(* IEC 61131-3 sources: Elmo_Master/test/Reports_Lasal/C78_20260807_publish_split_rebaseline (part 5) *)

	homePreemptionResult := CopyAxisOwnershipPreemption(
			PreemptedAdmissionToken:=homeAdmissionToken,
			PreemptedOwnerGeneration:=homeOwnerGeneration,
			pDest:=#homePreemptionSnapshot[0],
			DestSize:=sizeof(homePreemptionSnapshot));
	if (homePreemptionResult >= LMC_OWNER_PREEMPT_STATUS_PENDING_FREEZE) &
		   (homePreemptionResult <=
		    LMC_OWNER_PREEMPT_STATUS_CLEANUP_QUARANTINED) then
		homePreemptionSnapshotValid :=
				(homePreemptionSnapshot[0]$UDINT =
				 LMC_OWNER_PREEMPT_COPY_MAGIC) &
				(homePreemptionSnapshot[4]$UDINT =
				 LMC_OWNER_IDENTITY_VERSION) &
				(homePreemptionSnapshot[8]$UDINT =
				 LMC_OWNER_PREEMPT_COPY_HEADER_BYTES) &
				(homePreemptionSnapshot[12]$UDINT =
				 sizeof(homePreemptionSnapshot)) &
				(homePreemptionSnapshot[16]$DINT = homePreemptionResult) &
				(homePreemptionSnapshot[32]$UDINT =
				 homeAxisMask) &
				(homePreemptionSnapshot[36]$UDINT =
				 homeAdmissionToken) &
				(homePreemptionSnapshot[40]$UDINT =
				 homeOwnerGeneration) &
				(homePreemptionSnapshot[44]$UDINT =
				 homeSessionEpoch) &
				(homePreemptionSnapshot[48]$UDINT =
				 homeRequestSequence) &
				(homePreemptionSnapshot[52]$UDINT = 0x7D13) &
				(homePreemptionSnapshot[56]$DINT = ZeroHomeState[9]) &
				(homePreemptionSnapshot[60]$DINT =
				 LMC_OWNER_KIND_LMC_HOME) &
				(homePreemptionSnapshot[64]$DINT =
				 LMC_OWNER_RESOURCE_LMC_HOME_ENGINE) &
				(homePreemptionSnapshot[68]$DINT =
				 LMC_OWNER_ADMISSION_LIFECYCLE) &
				(homePreemptionSnapshot[72]$DINT =
				 LMC_OWNER_STATE_LMC_HOME_ACTIVE) &
				(homePreemptionSnapshot[76]$UDINT = 56) &
				((homePreemptionSnapshot[104]$UDINT and
				  homeAxisMask) = homeAxisMask) &
				(homePreemptionSnapshot[108]$UDINT <> 0) &
				(homePreemptionSnapshot[112]$UDINT <> 0) &
				((homePreemptionSnapshot[124]$DINT =
				  LMC_OWNER_STATE_RESERVED) |
				 (homePreemptionSnapshot[124]$DINT =
				  LMC_OWNER_STATE_SAFETY_PREEMPTING) |
				 (homePreemptionSnapshot[124]$DINT =
				  LMC_OWNER_STATE_QUARANTINED)) &
				(homePreemptionSnapshot[128]$UDINT <> 0) &
				(homePreemptionSnapshot[132]$UDINT <> 0) &
				(homePreemptionSnapshot[136]$DINT =
				 LMC_OWNER_ADMISSION_SAFETY) &
				(homePreemptionSnapshot[140]$UDINT = 0) &
				(homePreemptionSnapshot[144]$UINT = 1) &
				(homePreemptionSnapshot[146]$UINT = 0) &
				(homePreemptionSnapshot[148]$UDINT =
				 ZeroHomeState[4]$UDINT) &
				(homePreemptionSnapshot[152]$UDINT =
				 ZeroHomeState[1]$UDINT) &
				(homePreemptionSnapshot[156]$UDINT =
				 ZeroHomeState[2]$UDINT) &
				(homePreemptionSnapshot[160]$UDINT =
				 ZeroHomeState[3]$UDINT) &
				(homePreemptionSnapshot[164]$UDINT =
				 ZeroHomeState[5]$UDINT) &
				(homePreemptionSnapshot[168]$UDINT =
				 ZeroHomeState[6]$UDINT) &
				(homePreemptionSnapshot[172]$UDINT =
				 ZeroHomeState[7]$UDINT) &
				(homePreemptionSnapshot[176]$UDINT =
				 ZeroHomeState[8]$UDINT) &
				(homePreemptionSnapshot[180]$UINT =
				 TO_UINT(ZeroHomeState[10])) &
				(homePreemptionSnapshot[182]$UINT = 0) &
				(homePreemptionSnapshot[184]$DINT = ZeroHomeState[11]) &
				(homePreemptionSnapshot[188]$DINT = ZeroHomeState[12]) &
				(homePreemptionSnapshot[192]$UDINT =
				 ZeroHomeState[13]$UDINT) &
				(homePreemptionSnapshot[196]$UDINT = 0x454D4F48);
		if homePreemptionResult =
			   LMC_OWNER_PREEMPT_STATUS_PENDING_FREEZE then
			homePreemptionSnapshotValid :=
					homePreemptionSnapshotValid &
					((homePreemptionSnapshot[24]$UDINT and
					  homeAxisMask) = homeAxisMask) &
					((homePreemptionSnapshot[28]$UDINT and
					  homeAxisMask) = 0) &
					(homePreemptionSnapshot[124]$DINT =
					 LMC_OWNER_STATE_RESERVED);
		elsif homePreemptionResult =
			      LMC_OWNER_PREEMPT_STATUS_CLEANUP_REQUIRED then
			homePreemptionSnapshotValid :=
					homePreemptionSnapshotValid &
					((homePreemptionSnapshot[24]$UDINT and
					  homeAxisMask) = homeAxisMask) &
					((homePreemptionSnapshot[28]$UDINT and
					  homeAxisMask) = 0) &
					(homePreemptionSnapshot[124]$DINT <>
					 LMC_OWNER_STATE_RESERVED);
		elsif homePreemptionResult =
			      LMC_OWNER_PREEMPT_STATUS_CLEANUP_COMPLETE then
			homePreemptionSnapshotValid :=
					homePreemptionSnapshotValid &
					((homePreemptionSnapshot[28]$UDINT and
					  homeAxisMask) = homeAxisMask);
		end_if;
	end_if;

	if homePreemptionResult =
		   LMC_OWNER_PREEMPT_STATUS_PENDING_FREEZE then
		// The safety handler may run only after exact snapshot and cancel proof.
		homeFlags := homeFlags or LMC_HOME_FLAG_CANCEL_REQUIRED;
		ZeroHomeState[39] := LMC_HOME_ENGINE_CANCEL_DRAIN;
		if homePreemptionSnapshotValid &
		   (IsClientConnected(#InputLatch) <> 0) then
			homeCancelResult := InputLatch.CancelAxisZeroHome(
				OperationToken:=homeAdmissionToken);
		end_if;
		if homePreemptionSnapshotValid & (homeCancelResult >= 0) then
			if (homeFlags and LMC_HOME_FLAG_CANCEL_PUBLISHED) = 0 then
				ZeroHomeState[54]$UDINT := homeServiceNow;
			end_if;
			homeFlags := homeFlags or LMC_HOME_FLAG_CANCEL_PUBLISHED or
				LMC_HOME_FLAG_PREEMPTION_CLEANUP or
				LMC_HOME_FLAG_SAFETY_DISPATCH_READY;
		else
			ZeroHomeState[31] := homeCancelResult;
			OwnershipState[24] := 1;
		end_if;
		ZeroHomeState[56]$UDINT := homeFlags;
		RETURN;
	elsif (homePreemptionResult =
		       LMC_OWNER_PREEMPT_STATUS_CLEANUP_COMPLETE) &
		      homePreemptionSnapshotValid then
		// Exact owner cleanup replay is sufficient to finish the retained record.
		ZeroHomeState[14] := 1;
		ZeroHomeState[15] := -31000;
		ZeroHomeState[16] := 39;
		ZeroHomeState[30]$UDINT := homeServiceNow;
		ZeroHomeState[31] := -10;
		ZeroHomeState[47] := 1;
		ZeroHomeState[57] := LMC_HOME_RECORD_ABORTED;
		ZeroHomeState[58] := LMC_OWNER_REPORT_TERMINAL_SAFE_FAILURE;
		ZeroHomeState[59] := LMC_OWNER_CLEANUP_COMPLETE_SAFE;
		homeFlags := homeFlags or LMC_HOME_FLAG_CANCEL_REQUIRED or
			LMC_HOME_FLAG_CANCEL_PUBLISHED or
			LMC_HOME_FLAG_EXACT_RT_TERMINAL or
			LMC_HOME_FLAG_OWNER_FINALIZE_INTENT or
			LMC_HOME_FLAG_OWNER_FINALIZE_ACCEPTED or
			LMC_HOME_FLAG_TERMINAL_PUBLISHED or
			LMC_HOME_FLAG_PREEMPTION_CLEANUP;
		ZeroHomeState[56]$UDINT := homeFlags;
		ZeroHomeState[39] := LMC_HOME_ENGINE_TERMINAL;
		ZeroHomeState[0] := LMC_HOME_RECORD_ABORTED;
		RETURN;
	elsif (homePreemptionResult =
		       LMC_OWNER_PREEMPT_STATUS_CLEANUP_QUARANTINED) &
		      homePreemptionSnapshotValid then
		ZeroHomeState[14] := 1;
		ZeroHomeState[15] := -31000;
		ZeroHomeState[16] := 42;
		ZeroHomeState[30]$UDINT := homeServiceNow;
		ZeroHomeState[31] := -8;
		ZeroHomeState[47] := 1;
		ZeroHomeState[57] := LMC_HOME_RECORD_QUARANTINED;
		ZeroHomeState[58] := LMC_OWNER_REPORT_QUARANTINE;
		ZeroHomeState[59] := LMC_OWNER_CLEANUP_INCOMPLETE_QUARANTINE;
		homeFlags := homeFlags or LMC_HOME_FLAG_CANCEL_REQUIRED or
			LMC_HOME_FLAG_OWNER_FINALIZE_INTENT or
			LMC_HOME_FLAG_OWNER_FINALIZE_ACCEPTED or
			LMC_HOME_FLAG_TERMINAL_PUBLISHED or
			LMC_HOME_FLAG_PREEMPTION_CLEANUP;
		ZeroHomeState[56]$UDINT := homeFlags;
		ZeroHomeState[39] := LMC_HOME_ENGINE_TERMINAL;
		ZeroHomeState[0] := LMC_HOME_RECORD_QUARANTINED;
		RETURN;
	elsif (homePreemptionResult <> LMC_OWNER_PREEMPT_STATUS_NONE) &
		      ((homePreemptionResult <
		        LMC_OWNER_PREEMPT_STATUS_PENDING_FREEZE) |
		       (homePreemptionResult >
		        LMC_OWNER_PREEMPT_STATUS_CLEANUP_QUARANTINED) |
		       (homePreemptionSnapshotValid = FALSE)) then
		homeFlags := homeFlags or LMC_HOME_FLAG_CANCEL_REQUIRED;
		ZeroHomeState[39] := LMC_HOME_ENGINE_CANCEL_DRAIN;
		if IsClientConnected(#InputLatch) <> 0 then
			homeCancelResult := InputLatch.CancelAxisZeroHome(
				OperationToken:=homeAdmissionToken);
			if homeCancelResult >= 0 then
				if (homeFlags and LMC_HOME_FLAG_CANCEL_PUBLISHED) = 0 then
					ZeroHomeState[54]$UDINT := homeServiceNow;
				end_if;
				homeFlags := homeFlags or LMC_HOME_FLAG_CANCEL_PUBLISHED;
			end_if;
		end_if;
		ZeroHomeState[31] := homePreemptionResult;
		ZeroHomeState[56]$UDINT := homeFlags;
		OwnershipState[24] := 1;
		RETURN;
	elsif homePreemptionResult =
		      LMC_OWNER_PREEMPT_STATUS_CLEANUP_REQUIRED then
		homePreemptionCleanup := TRUE;
		homeCancelRequired := TRUE;
		homeFlags := homeFlags or LMC_HOME_FLAG_CANCEL_REQUIRED or
			LMC_HOME_FLAG_PREEMPTION_CLEANUP;
		if homeEngineState <> LMC_HOME_ENGINE_FINALIZE then
			ZeroHomeState[39] := LMC_HOME_ENGINE_CANCEL_DRAIN;
		end_if;
	elsif homePreemptionResult = LMC_OWNER_PREEMPT_STATUS_NONE then
		if homePreemptionCleanup then
			// A rejected safety reservation restored the old Home owner.
			homePreemptionCleanup := FALSE;
			homeFlags := homeFlags and 0xFFFFFF7F;
		end_if;
		if homeEngineState = LMC_HOME_ENGINE_WAIT_RT then
			homeOwnerResult := ValidateAxisOwnership(
				CommandId:=0x7D13,
				Reference:=ZeroHomeState[9]$UINT,
				ExpectedAxisMask:=homeAxisMask,
				OwnerKind:=LMC_OWNER_KIND_LMC_HOME,
				ResourceKind:=LMC_OWNER_RESOURCE_LMC_HOME_ENGINE,
				AdmissionMode:=LMC_OWNER_ADMISSION_LIFECYCLE,
				CallerSessionEpoch:=homeSessionEpoch,
				RequestSequence:=homeRequestSequence,
				AdmissionToken:=homeAdmissionToken,
				OwnerGeneration:=homeOwnerGeneration,
				RequiredPhase:=LMC_OWNER_PHASE_ACTIVE);
			if homeOwnerResult <> 0 then
				homeCancelRequired := TRUE;
				homeFlags := homeFlags or LMC_HOME_FLAG_CANCEL_REQUIRED;
				ZeroHomeState[31] := homeOwnerResult;
				ZeroHomeState[39] := LMC_HOME_ENGINE_CANCEL_DRAIN;
				OwnershipState[24] := 1;
			elsif IsClientConnected(#InputLatch) = 0 then
				homeCancelRequired := TRUE;
				homeFlags := homeFlags or LMC_HOME_FLAG_CANCEL_REQUIRED;
				ZeroHomeState[31] := -3;
				ZeroHomeState[39] := LMC_HOME_ENGINE_CANCEL_DRAIN;
				OwnershipState[24] := 1;
			end_if;
		end_if;
	else
		OwnershipState[24] := 1;
		RETURN;
	end_if;

	if homeEngineState = LMC_HOME_ENGINE_FINALIZE then
		homePendingRecordState := ZeroHomeState[57];
		homeReportKind := ZeroHomeState[58]$UINT;
		homeCleanupKind := ZeroHomeState[59]$UINT;
		homeReceiptRequired :=
			(homePreemptionCleanup = FALSE) &
			(homePendingRecordState <> LMC_HOME_RECORD_QUARANTINED) &
			((homeReportKind = LMC_OWNER_REPORT_TERMINAL_SUCCESS) |
			 (homeReportKind = LMC_OWNER_REPORT_TERMINAL_SAFE_FAILURE));
		if (homePendingRecordState < LMC_HOME_RECORD_SUCCEEDED) |
		   (homePendingRecordState > LMC_HOME_RECORD_QUARANTINED) |
		   (homeReportKind < LMC_OWNER_REPORT_TERMINAL_SUCCESS) |
		   (homeReportKind > LMC_OWNER_REPORT_QUARANTINE) |
		   ((homeFlags and LMC_HOME_FLAG_OWNER_FINALIZE_INTENT) = 0) |
		   ((homeReceiptRequired = FALSE) &
		    ((ZeroHomeState[60] <> 0) | (ZeroHomeState[61] <> 0) |
		     (ZeroHomeState[62] <> 0) | (ZeroHomeState[63] <> 0))) then
			OwnershipState[24] := 1;
			RETURN;
		end_if;
		if (homeFlags and LMC_HOME_FLAG_OWNER_FINALIZE_ACCEPTED) = 0 then
			if homePreemptionCleanup then
				if (homePreemptionResult <>
				    LMC_OWNER_PREEMPT_STATUS_CLEANUP_REQUIRED) |
				   (homePreemptionSnapshotValid = FALSE) then
					OwnershipState[24] := 1;
					RETURN;
				end_if;
				homePublishResult := PublishAxisOwnershipPreemptionCleanup(
					ExpectedAxisMask:=homeAxisMask,
					PreemptedAdmissionToken:=homeAdmissionToken,
					PreemptedOwnerGeneration:=homeOwnerGeneration,
					SafetyAdmissionToken:=homePreemptionSnapshot[108]$UDINT,
					SafetyOwnerGeneration:=homePreemptionSnapshot[112]$UDINT,
					CleanupKind:=homeCleanupKind,
					ReportValue0:=TO_UDINT(homePendingRecordState),
					ReportValue1:=ZeroHomeState[31]$UDINT,
					ObservationCycle:=ZeroHomeState[46]$UDINT);
			else
				if homePreemptionResult <> LMC_OWNER_PREEMPT_STATUS_NONE then
					OwnershipState[24] := 1;
					RETURN;
				end_if;
				homePublishResult := PublishAxisOwnership(
					AxisMask:=homeAxisMask,
					AdmissionToken:=homeAdmissionToken,
					OwnerGeneration:=homeOwnerGeneration,
					ReportKind:=homeReportKind,
					ReportValue0:=TO_UDINT(homePendingRecordState),
					ReportValue1:=ZeroHomeState[31]$UDINT,
					ObservationCycle:=ZeroHomeState[46]$UDINT);
			end_if;
			ZeroHomeState[47] := homePublishResult;
			if homeReceiptRequired then
				if (homePublishResult <> 0) |
				   (ZeroHomeState[60]$UDINT <>
				    LMC_HOME_OWNER_RECEIPT_MAGIC) |
				   (ZeroHomeState[61] <>
				    LMC_HOME_OWNER_RECEIPT_PREPARED) |
				   (ZeroHomeState[62] <> 0) |
				   (ZeroHomeState[63]$UDINT <>
				    ZeroHomeState[33]$UDINT) then
					OwnershipState[24] := 1;
					RETURN;
				end_if;
			elsif (homePublishResult <> 0) & (homePublishResult <> 1) then
				OwnershipState[24] := 1;
				RETURN;
			end_if;
			homeFlags := homeFlags or LMC_HOME_FLAG_OWNER_FINALIZE_ACCEPTED;
			ZeroHomeState[56]$UDINT := homeFlags;
		end_if;
		if homeReceiptRequired then
			if (ZeroHomeState[60]$UDINT <>
			    LMC_HOME_OWNER_RECEIPT_MAGIC) |
			   (ZeroHomeState[62] <> 0) |
			   (ZeroHomeState[63]$UDINT <> ZeroHomeState[33]$UDINT) then
				OwnershipState[24] := 1;
				RETURN;
			end_if;
			homePublishResult := PublishAxisOwnership(
				AxisMask:=homeAxisMask,
				AdmissionToken:=homeAdmissionToken,
				OwnerGeneration:=homeOwnerGeneration,
				ReportKind:=homeReportKind,
				ReportValue0:=TO_UDINT(homePendingRecordState),
				ReportValue1:=ZeroHomeState[31]$UDINT,
				ObservationCycle:=ZeroHomeState[46]$UDINT);
			ZeroHomeState[47] := homePublishResult;
			if homePublishResult = LMC_OWNER_REBASE_PERSIST_RETRY then
				// Keep FINALIZE and retry the retained barrier write next cycle.
				// Global owner quarantine would block the Home recovery path itself.
				RETURN;
			end_if;
			if (homePublishResult <> 1) |
			   (ZeroHomeState[61] <>
			    LMC_HOME_OWNER_RECEIPT_COMPLETE) then
				OwnershipState[24] := 1;
				RETURN;
			end_if;
		end_if;
		homeFlags := homeFlags or LMC_HOME_FLAG_TERMINAL_PUBLISHED;
		ZeroHomeState[56]$UDINT := homeFlags;
		ZeroHomeState[39] := LMC_HOME_ENGINE_TERMINAL;
		ZeroHomeState[0] := homePendingRecordState;
		RETURN;
	end_if;

	if homeCancelRequired |
	   (ZeroHomeState[39] = LMC_HOME_ENGINE_CANCEL_DRAIN) then
		homeFlags := homeFlags or LMC_HOME_FLAG_CANCEL_REQUIRED;
		ZeroHomeState[39] := LMC_HOME_ENGINE_CANCEL_DRAIN;
		if IsClientConnected(#InputLatch) <> 0 then
			homeCancelResult := InputLatch.CancelAxisZeroHome(
				OperationToken:=homeAdmissionToken);
		end_if;
		if homeCancelResult < 0 then
			ZeroHomeState[31] := homeCancelResult;
			ZeroHomeState[56]$UDINT := homeFlags;
			OwnershipState[24] := 1;
			RETURN;
		end_if;
		if (homeFlags and LMC_HOME_FLAG_CANCEL_PUBLISHED) = 0 then
			ZeroHomeState[54]$UDINT := homeServiceNow;
			homeCancelElapsedMs := 0;
		end_if;
		homeFlags := homeFlags or LMC_HOME_FLAG_CANCEL_PUBLISHED;
		ZeroHomeState[56]$UDINT := homeFlags;
	end_if;

	if IsClientConnected(#InputLatch) = 0 then
		ZeroHomeState[31] := -3;
		OwnershipState[24] := 1;
		RETURN;
	end_if;
	homeCopyResult := InputLatch.CopyAxisZeroHomeResult(
		OperationToken:=homeAdmissionToken,
		pDest:=#homeLatchResult[0],
		DestSize:=128);

	if homeCopyResult = 0 then
			homeNativeCallCount := homeLatchResult[8];
			homeObservationCycle := homeLatchResult[23]$UDINT;
			if (homeLatchResult[0]$UDINT <> homeAdmissionToken) |
			   (homeLatchResult[3] <> ZeroHomeState[9]) |
			   (homeLatchResult[4] <> ZeroHomeState[11]) |
			   (homeLatchResult[22]$UDINT = 0) |
			   ((homeLatchResult[1] <> LMC_HOME_RECORD_SUCCEEDED) &
			    (homeLatchResult[1] <> LMC_HOME_RECORD_FAILED)) then
				homeFailureCode := -8;
				homeQuarantine := TRUE;
			elsif (homeLatchResult[1] = LMC_HOME_RECORD_SUCCEEDED) &
			      (homeLatchResult[2] = 0) &
			      (homeLatchResult[6] = 3) &
			      (homeLatchResult[7]$UDINT = LMC_HOME_EVIDENCE_COMPLETE) &
			      (homeLatchResult[8] = 1) &
			      (homeLatchResult[10]$UDINT <> 0) &
			      ((homeLatchResult[11]$UDINT and
			        LMC_AXIS_STATUS_STANDSTILL) <> 0) &
			      (homeLatchResult[12] = 0) &
			      (homeLatchResult[15] = 0) &
			      (homeLatchResult[16] = 0) &
			      (homeLatchResult[17] = 0) &
			      (homeLatchResult[18] = 0) &
			      (homeLatchResult[19] = 0) &
			      (homeLatchResult[20] = 0) &
			      (homeLatchResult[21] = 0) &
			      (ZeroHomeState[53] = 0) then
				homeSucceeded := TRUE;
				homeExactRtTerminal := TRUE;
			elsif homeLatchResult[1] = LMC_HOME_RECORD_FAILED then
				homeFailureCode := homeLatchResult[2];
				if homeFailureCode = 0 then
					homeFailureCode := -8;
				else
					homeExactRtTerminal := TRUE;
				end_if;
				if homeFailureCode = -10 then
					homeAborted := TRUE;
				end_if;
				if homeNativeCallCount <> 0 then
					homeQuarantine := TRUE;
				end_if;
			else
				homeFailureCode := -8;
				homeQuarantine := TRUE;
			end_if;
			homeTerminal := TRUE;
	elsif homeCopyResult = 1 then
		if ((homeFlags and LMC_HOME_FLAG_CANCEL_PUBLISHED) <> 0) &
		   (homeCancelElapsedMs >= LMC_HOME_CANCEL_DRAIN_TIMEOUT_MS) then
			homeFailureCode := -10;
			homeQuarantine := TRUE;
			homeTerminal := TRUE;
		elsif (homeFlags and LMC_HOME_FLAG_CANCEL_REQUIRED) = 0 then
			if homeElapsedMs >= ZeroHomeState[13]$UDINT then
			homeCancelResult := InputLatch.CancelAxisZeroHome(
				OperationToken:=homeAdmissionToken);
				homeFlags := homeFlags or LMC_HOME_FLAG_CANCEL_REQUIRED;
				ZeroHomeState[39] := LMC_HOME_ENGINE_CANCEL_DRAIN;
				if homeCancelResult >= 0 then
					ZeroHomeState[54]$UDINT := homeServiceNow;
					homeFlags := homeFlags or LMC_HOME_FLAG_CANCEL_PUBLISHED;
				else
					ZeroHomeState[31] := homeCancelResult;
					OwnershipState[24] := 1;
				end_if;
				ZeroHomeState[56]$UDINT := homeFlags;
			end_if;
		end_if;
	else
		ZeroHomeState[31] := homeCopyResult;
		ZeroHomeState[56]$UDINT := homeFlags or
			LMC_HOME_FLAG_CANCEL_REQUIRED;
		ZeroHomeState[39] := LMC_HOME_ENGINE_CANCEL_DRAIN;
		OwnershipState[24] := 1;
		RETURN;
	end_if;

	if homeTerminal = FALSE then
		RETURN;
	end_if;

	if homeObservationCycle = 0 then
		homeObservationCycle := homeServiceNow;
	end_if;
	ZeroHomeState[17]$UDINT := homeLatchResult[11]$UDINT;
	ZeroHomeState[18] := homeLatchResult[12];
	ZeroHomeState[19] := homeLatchResult[13];
	ZeroHomeState[20] := homeLatchResult[14];
	ZeroHomeState[21] := homeLatchResult[15];
	ZeroHomeState[22] := homeLatchResult[16];
	ZeroHomeState[23] := homeLatchResult[17];
	ZeroHomeState[24] := homeLatchResult[18];
	ZeroHomeState[25] := homeLatchResult[19];
	ZeroHomeState[26] := homeLatchResult[20];
	ZeroHomeState[27]$UDINT := homeLatchResult[21]$UDINT;
	ZeroHomeState[28]$UDINT := homeLatchResult[7]$UDINT;
	ZeroHomeState[30]$UDINT := homeServiceNow;
	ZeroHomeState[31] := homeFailureCode;
	ZeroHomeState[32] := homeLatchResult[5];
	ZeroHomeState[40] := homeLatchResult[1];
	ZeroHomeState[41] := homeFailureCode;
	ZeroHomeState[42] := homeNativeCallCount;
	ZeroHomeState[43] := homeLatchResult[6];
	ZeroHomeState[44]$UDINT := homeLatchResult[9]$UDINT;
	ZeroHomeState[45]$UDINT := homeLatchResult[10]$UDINT;
	ZeroHomeState[46]$UDINT := homeObservationCycle;
	ZeroHomeState[55]$UDINT := homeLatchResult[22]$UDINT;

	if homeSucceeded then
		homePendingRecordState := LMC_HOME_RECORD_SUCCEEDED;
		ZeroHomeState[14] := 0;
		ZeroHomeState[15] := 0;
		ZeroHomeState[16] := 0;
		ZeroHomeState[31] := 0;
		homeReportKind := LMC_OWNER_REPORT_TERMINAL_SUCCESS;
	elsif homeQuarantine then
		homePendingRecordState := LMC_HOME_RECORD_QUARANTINED;
		ZeroHomeState[14] := 1;
		ZeroHomeState[15] := -31000;
		if homeAborted then
			ZeroHomeState[16] := 39;
		elsif homePreemptionResult <> LMC_OWNER_PREEMPT_STATUS_NONE then
			ZeroHomeState[16] := 42;
		else
			ZeroHomeState[16] := 38;
		end_if;
		homeReportKind := LMC_OWNER_REPORT_QUARANTINE;
	elsif homeAborted then
		homePendingRecordState := LMC_HOME_RECORD_ABORTED;
		ZeroHomeState[14] := 1;
		ZeroHomeState[15] := -31000;
		ZeroHomeState[16] := 39;
		homeReportKind := LMC_OWNER_REPORT_TERMINAL_SAFE_FAILURE;
	else
		homePendingRecordState := LMC_HOME_RECORD_FAILED;
		ZeroHomeState[14] := 1;
		ZeroHomeState[15] := -31000;
		ZeroHomeState[16] := 38;
		homeReportKind := LMC_OWNER_REPORT_TERMINAL_SAFE_FAILURE;
	end_if;

	if homePreemptionCleanup then
		if homeExactRtTerminal then
			if homeQuarantine then
				homeCleanupKind := LMC_OWNER_CLEANUP_COMPLETE_QUARANTINE;
			else
				homeCleanupKind := LMC_OWNER_CLEANUP_COMPLETE_SAFE;
			end_if;
		else
			homeCleanupKind := LMC_OWNER_CLEANUP_INCOMPLETE_QUARANTINE;
		end_if;
	else
		homeCleanupKind := 0;
	end_if;
	if homeExactRtTerminal then
		homeFlags := homeFlags or LMC_HOME_FLAG_EXACT_RT_TERMINAL;
	end_if;
	homeFlags := homeFlags or LMC_HOME_FLAG_OWNER_FINALIZE_INTENT;
	ZeroHomeState[56]$UDINT := homeFlags;
	ZeroHomeState[57] := homePendingRecordState;
	ZeroHomeState[58] := TO_DINT(homeReportKind);
	ZeroHomeState[59] := TO_DINT(homeCleanupKind);
	ZeroHomeState[39] := LMC_HOME_ENGINE_FINALIZE;

END_FUNCTION

FUNCTION LMCControlCommandService::HandleAxisZeroHomeCommands
	VAR_INPUT
		CommandId 	: UINT;
		Reference 	: UINT;
		pRequestFrame 	: ^USINT;
		RequestFrameSize 	: UDINT;
		pResponseFrame 	: ^USINT;
		ResponseCapacity 	: UDINT;
	END_VAR
	VAR_OUTPUT
		ResponseSize 	: DINT;
	END_VAR
	VAR
		pRequest : ^USINT;
		RequestSize : UDINT;
		adminSchemaVersion : UINT;
		adminRequestFlags : UINT;
		adminRequestId : UDINT;
		adminDiagnosticsBuild : UDINT;
		adminBootId : UDINT;
		adminMapRevision : UDINT;
		adminClientIntentId0 : UDINT;
		adminClientIntentId1 : UDINT;
		adminClientIntentId2 : UDINT;
		adminClientIntentId3 : UDINT;
		adminCurrentBootId : UDINT;
		adminOriginalRequestId : UDINT;
		adminDetailCode : UDINT;
		adminHomeSemanticMode : UINT;
		adminHomeReserved : UINT;
		adminHomeExpectedActualPosition : DINT;
		adminHomeTargetPosition : DINT;
		adminHomeTimeoutMs : UDINT;
		adminHomeExecuteToken : UDINT;
		adminHomeRecordGeneration : UDINT;
		adminHomeAxisMask : UDINT;
		adminHomeServiceNow : UDINT;
		adminHomeStateIndex : DINT;
		adminHomeSubmitResult : DINT;
		adminHomeOwnerResult : DINT;
		adminHomeRecordState : DINT;
		adminHomeGenerationCounter : UDINT;
		adminHomeRecordValid : BOOL;
		adminHomeIdentityValid : BOOL;
		adminHomeTerminal : BOOL;
		adminHomeEmptyValid : BOOL;
		adminHomeStateConsistent : BOOL;
		adminErrorId : INT;
	END_VAR

	ResponseSize := -1;
	if (pRequestFrame = NIL) | (pResponseFrame = NIL) |
	   (RequestFrameSize < 8) then
		RETURN;
	end_if;
	pRequest := pRequestFrame + 8;
	RequestSize := RequestFrameSize - 8;

	case CommandId of
		// LMC_Home only rebases the current coordinate through the RT mailbox.
		0x7D13:
			if ResponseCapacity < 32 then
				RETURN;
			end_if;
			adminSchemaVersion := 0;
			adminRequestFlags := 0;
			adminRequestId := 0;
			adminDiagnosticsBuild := 0;
			adminBootId := 0;
			adminMapRevision := 0;
			adminClientIntentId0 := 0;
			adminClientIntentId1 := 0;
			adminClientIntentId2 := 0;
			adminClientIntentId3 := 0;
			adminHomeSemanticMode := 0;
			adminHomeReserved := 0;
			adminHomeExpectedActualPosition := 0;
			adminHomeTargetPosition := 0;
			adminHomeTimeoutMs := 0;
			adminHomeExecuteToken := 0;
			adminHomeAxisMask := 0;
			adminHomeSubmitResult := -1;
			adminHomeOwnerResult := -1;
			adminDetailCode := 0;
			adminErrorId := -31000;

			if RequestSize >= 8 then
				adminSchemaVersion := pRequest^$UINT;
				adminRequestFlags := (pRequest + 2)^$UINT;
				adminRequestId := (pRequest + 4)^$UDINT;
			end_if;
			if RequestSize >= 56 then
				adminDiagnosticsBuild := (pRequest + 8)^$UDINT;
				adminBootId := (pRequest + 12)^$UDINT;
				adminMapRevision := (pRequest + 16)^$UDINT;
				adminClientIntentId0 := (pRequest + 20)^$UDINT;
				adminClientIntentId1 := (pRequest + 24)^$UDINT;
				adminClientIntentId2 := (pRequest + 28)^$UDINT;
				adminClientIntentId3 := (pRequest + 32)^$UDINT;
				adminHomeSemanticMode := (pRequest + 36)^$UINT;
				adminHomeReserved := (pRequest + 38)^$UINT;
				adminHomeExpectedActualPosition := (pRequest + 40)^$DINT;
				adminHomeTargetPosition := (pRequest + 44)^$DINT;
				adminHomeTimeoutMs := (pRequest + 48)^$UDINT;
				adminHomeExecuteToken := (pRequest + 52)^$UDINT;
			end_if;

			case Reference of
				1: adminHomeAxisMask := 0x00000001;
				2: adminHomeAxisMask := 0x00000002;
				3: adminHomeAxisMask := 0x00000004;
				4: adminHomeAxisMask := 0x00000008;
			else
			end_case;

			adminHomeRecordState := ZeroHomeState[0];
			adminHomeRecordValid :=
				(ZeroHomeState[51]$UDINT = LMC_HOME_RECORD_MAGIC) &
				(ZeroHomeState[33]$UDINT <> 0);
			adminHomeTerminal :=
				(adminHomeRecordState >= LMC_HOME_RECORD_SUCCEEDED) &
				(adminHomeRecordState <= LMC_HOME_RECORD_QUARANTINED);
			adminHomeEmptyValid := TRUE;
			if adminHomeRecordState = LMC_HOME_RECORD_EMPTY then
				adminHomeStateIndex := 1;
				while adminHomeStateIndex <= 63 do
					if (adminHomeStateIndex <> 50) &
					   (ZeroHomeState[adminHomeStateIndex] <> 0) then
						adminHomeEmptyValid := FALSE;
					end_if;
					adminHomeStateIndex += 1;
				end_while;
			end_if;

			if RequestSize <> 56 then
				adminDetailCode := 5;
			elsif (Reference < 1) | (Reference > 4) then
				adminDetailCode := 4;
			elsif adminSchemaVersion <> 1 then
				adminDetailCode := 1;
			elsif adminRequestFlags <> 0 then
				adminDetailCode := 2;
			elsif adminRequestId = 0 then
				adminDetailCode := 3;
			elsif adminDiagnosticsBuild = 0 then
				adminDetailCode := 16;
			elsif adminBootId = 0 then
				adminDetailCode := 17;
			elsif adminMapRevision = 0 then
				adminDetailCode := 18;
			elsif (adminClientIntentId0 = 0) &
			      (adminClientIntentId1 = 0) &
			      (adminClientIntentId2 = 0) &
			      (adminClientIntentId3 = 0) then
				adminDetailCode := 15;
			elsif (adminHomeSemanticMode <> 1) |
			      (adminHomeReserved <> 0) |
			      (adminHomeTargetPosition <> 0) |
			      (adminHomeTimeoutMs < 100) |
			      (adminHomeTimeoutMs > 5000) |
			      (adminHomeExecuteToken <> 0x454D4F48) then
				adminDetailCode := 15;
			elsif LMC_ADMIN_AXIS_HOME_ENABLED = FALSE then
				adminDetailCode := 10;
			elsif IsClientConnected(#InputLatch) = 0 then
				adminDetailCode := 42;
			elsif (OwnershipState[0]$UDINT <> LMC_OWNER_TABLE_MAGIC) |
			      (OwnershipState[3]$UDINT = 0) then
				adminDetailCode := 42;
			elsif adminBootId <> OwnershipState[3]$UDINT then
				adminDetailCode := 17;
			elsif (adminHomeRecordState = LMC_HOME_RECORD_EMPTY) &
			      (adminHomeEmptyValid = FALSE) then
				adminDetailCode := 42;
			elsif (adminHomeRecordState <> LMC_HOME_RECORD_EMPTY) &
			      (adminHomeRecordValid = FALSE) then
				adminDetailCode := 42;
			elsif (adminHomeRecordState <> LMC_HOME_RECORD_EMPTY) &
			      ((adminHomeTerminal = FALSE) |
			       (adminHomeRecordState = LMC_HOME_RECORD_QUARANTINED) |
			       (ZeroHomeState[39] <> LMC_HOME_ENGINE_TERMINAL) |
			       ((ZeroHomeState[56]$UDINT and
			         LMC_HOME_FLAG_EXACT_RT_TERMINAL) = 0) |
			       ((ZeroHomeState[56]$UDINT and
			         LMC_HOME_FLAG_OWNER_FINALIZE_ACCEPTED) = 0) |
			       ((ZeroHomeState[56]$UDINT and
			         LMC_HOME_FLAG_TERMINAL_PUBLISHED) = 0) |
			       ((ZeroHomeState[47] <> 0) & (ZeroHomeState[47] <> 1)) |
			       (((ZeroHomeState[56]$UDINT and
			          LMC_HOME_FLAG_PREEMPTION_CLEANUP) = 0) &
			        (ZeroHomeState[47] <> 1)) |
			       (((ZeroHomeState[56]$UDINT and
			          LMC_HOME_FLAG_PREEMPTION_CLEANUP) = 0) &
			        ((ZeroHomeState[60]$UDINT <>
			          LMC_HOME_OWNER_RECEIPT_MAGIC) |
			         (ZeroHomeState[61] <>
			          LMC_HOME_OWNER_RECEIPT_COMPLETE) |
			         (ZeroHomeState[62] <> 0) |
			         (ZeroHomeState[63]$UDINT <>
			          ZeroHomeState[33]$UDINT))) |
			       (ZeroHomeState[48] = 0) |
			       (ZeroHomeState[49]$UDINT <> ZeroHomeState[33]$UDINT)) then
				adminDetailCode := 40;
			else
				adminHomeOwnerResult := ValidateAxisOwnershipIdentity(
					CommandId:=0x7D13,
					Reference:=Reference,
					ExpectedAxisMask:=adminHomeAxisMask,
					OwnerKind:=LMC_OWNER_KIND_LMC_HOME,
					ResourceKind:=LMC_OWNER_RESOURCE_LMC_HOME_ENGINE,
					AdmissionMode:=LMC_OWNER_ADMISSION_LIFECYCLE,
					CallerSessionEpoch:=OwnershipState[16]$UDINT,
					RequestSequence:=OwnershipState[17]$UDINT,
					AdmissionToken:=OwnershipState[18]$UDINT,
					OwnerGeneration:=OwnershipState[19]$UDINT,
					RequiredPhase:=LMC_OWNER_PHASE_RESERVED,
					pIdentity:=pRequest$^void,
					IdentitySize:=RequestSize);
				if adminHomeOwnerResult = -3 then
					adminDetailCode := 42;
				elsif adminHomeOwnerResult <> 0 then
					adminDetailCode := 41;
				else
					adminHomeGenerationCounter := ZeroHomeState[50]$UDINT + 1;
					if adminHomeGenerationCounter = 0 then
						adminHomeGenerationCounter := 1;
					end_if;
					_memset(dest:=#ZeroHomeState[0], usByte:=0, cntr:=256);
					ZeroHomeState[0] := LMC_HOME_RECORD_RUNNING;
					ZeroHomeState[1]$UDINT := adminDiagnosticsBuild;
					ZeroHomeState[2]$UDINT := adminBootId;
					ZeroHomeState[3]$UDINT := adminMapRevision;
					ZeroHomeState[4]$UDINT := adminRequestId;
					ZeroHomeState[5]$UDINT := adminClientIntentId0;
					ZeroHomeState[6]$UDINT := adminClientIntentId1;
					ZeroHomeState[7]$UDINT := adminClientIntentId2;
					ZeroHomeState[8]$UDINT := adminClientIntentId3;
					ZeroHomeState[9] := TO_DINT(Reference);
					ZeroHomeState[10] := TO_DINT(adminHomeSemanticMode);
					ZeroHomeState[11] := adminHomeExpectedActualPosition;
					ZeroHomeState[12] := adminHomeTargetPosition;
					ZeroHomeState[13]$UDINT := adminHomeTimeoutMs;
					ZeroHomeState[14] := 0;
					ZeroHomeState[15] := 0;
					ZeroHomeState[16] := 0;
					adminHomeServiceNow := ops.tAbsolute;
					if adminHomeServiceNow = 0 then
						adminHomeServiceNow := 1;
					end_if;
					ZeroHomeState[29]$UDINT := adminHomeServiceNow;
					ZeroHomeState[33]$UDINT := adminHomeGenerationCounter;
					ZeroHomeState[34]$UDINT := OwnershipState[18]$UDINT;
					ZeroHomeState[35]$UDINT := OwnershipState[19]$UDINT;
					ZeroHomeState[36]$UDINT := OwnershipState[16]$UDINT;
					ZeroHomeState[37]$UDINT := OwnershipState[17]$UDINT;
					ZeroHomeState[38]$UDINT := adminHomeAxisMask;
					ZeroHomeState[39] := LMC_HOME_ENGINE_WAIT_RT;
					ZeroHomeState[50]$UDINT := adminHomeGenerationCounter;
					ZeroHomeState[51]$UDINT := LMC_HOME_RECORD_MAGIC;

					adminHomeSubmitResult := InputLatch.SubmitAxisZeroHome(
						OperationToken:=OwnershipState[18]$UDINT,
						AxisReference:=TO_DINT(Reference),
						ExpectedActualPosition:=adminHomeExpectedActualPosition);
					ZeroHomeState[52] := adminHomeSubmitResult;
					if adminHomeSubmitResult = 1 then
						adminHomeOwnerResult := CommitAxisOwnership(
							CommandId:=0x7D13,
							Reference:=Reference,
							ExpectedAxisMask:=adminHomeAxisMask,
							CallerSessionEpoch:=OwnershipState[16]$UDINT,
							RequestSequence:=OwnershipState[17]$UDINT,
							AdmissionToken:=OwnershipState[18]$UDINT,
							OwnerGeneration:=OwnershipState[19]$UDINT);
						ZeroHomeState[47] := adminHomeOwnerResult;
						if adminHomeOwnerResult <> 0 then
							// The mailbox boundary was crossed; retain and quarantine later.
							ZeroHomeState[53] := 1;
						end_if;
						adminErrorId := 0;
					else
						adminHomeGenerationCounter := ZeroHomeState[50]$UDINT;
						_memset(dest:=#ZeroHomeState[0], usByte:=0, cntr:=256);
						ZeroHomeState[50]$UDINT := adminHomeGenerationCounter;
						if adminHomeSubmitResult = -2 then
							adminDetailCode := 41;
						else
							adminDetailCode := 42;
						end_if;
					end_if;
				end_if;
			end_if;

			if adminErrorId = 0 then
				_memset(dest:=pResponseFrame, usByte:=0, cntr:=32);
				pResponseFrame^$UINT := 0;
				(pResponseFrame + 2)^$UINT := 24;
				(pResponseFrame + 4)^$UDINT := 0;
				(pResponseFrame + 8)^$UINT := 1;
				(pResponseFrame + 10)^$UINT := 0;
				(pResponseFrame + 12)^$UINT := 0;
				(pResponseFrame + 14)^$INT := 0;
				(pResponseFrame + 16)^$UDINT := adminRequestId;
				(pResponseFrame + 20)^$UDINT := 0;
				(pResponseFrame + 24)^$UINT := adminHomeSemanticMode;
				(pResponseFrame + 26)^$UINT := 0;
				(pResponseFrame + 28)^$UDINT := 0;
				ResponseSize := 32;
			else
				_memset(dest:=pResponseFrame, usByte:=0, cntr:=24);
				pResponseFrame^$UINT := 0;
				(pResponseFrame + 2)^$UINT := 16;
				(pResponseFrame + 4)^$UDINT := 0;
				(pResponseFrame + 8)^$UINT := 1;
				(pResponseFrame + 10)^$UINT := 0;
				(pResponseFrame + 12)^$UINT := 1;
				(pResponseFrame + 14)^$INT := -31000;
				(pResponseFrame + 16)^$UDINT := adminRequestId;
				(pResponseFrame + 20)^$UDINT := adminDetailCode;
				ResponseSize := 24;
			end_if;

		0x7D18:
			if ResponseCapacity < 152 then
				RETURN;
			end_if;
			adminDetailCode := 0;
			adminSchemaVersion := 0;
			adminRequestFlags := 0;
			adminRequestId := 0;
			adminDiagnosticsBuild := 0;
			adminBootId := 0;
			adminMapRevision := 0;
			adminCurrentBootId := 0;
			adminOriginalRequestId := 0;
			adminClientIntentId0 := 0;
			adminClientIntentId1 := 0;
			adminClientIntentId2 := 0;
			adminClientIntentId3 := 0;
			adminHomeSemanticMode := 0;
			adminHomeReserved := 0;
			adminHomeExpectedActualPosition := 0;
			adminHomeTargetPosition := 0;
			adminHomeAxisMask := 0;
			if RequestSize >= 8 then
				adminSchemaVersion := pRequest^$UINT;
				adminRequestFlags := (pRequest + 2)^$UINT;
				adminRequestId := (pRequest + 4)^$UDINT;
			end_if;
			if RequestSize >= 56 then
				adminDiagnosticsBuild := (pRequest + 8)^$UDINT;
				adminBootId := (pRequest + 12)^$UDINT;
				adminMapRevision := (pRequest + 16)^$UDINT;
				adminCurrentBootId := (pRequest + 20)^$UDINT;
				adminOriginalRequestId := (pRequest + 24)^$UDINT;
				adminClientIntentId0 := (pRequest + 28)^$UDINT;
				adminClientIntentId1 := (pRequest + 32)^$UDINT;
				adminClientIntentId2 := (pRequest + 36)^$UDINT;
				adminClientIntentId3 := (pRequest + 40)^$UDINT;
				adminHomeSemanticMode := (pRequest + 44)^$UINT;
				adminHomeReserved := (pRequest + 46)^$UINT;
				adminHomeExpectedActualPosition := (pRequest + 48)^$DINT;
				adminHomeTargetPosition := (pRequest + 52)^$DINT;
			end_if;
			case Reference of
				1: adminHomeAxisMask := 0x00000001;
				2: adminHomeAxisMask := 0x00000002;
				3: adminHomeAxisMask := 0x00000004;
				4: adminHomeAxisMask := 0x00000008;
			else
			end_case;
			adminHomeRecordValid :=
				(ZeroHomeState[51]$UDINT = LMC_HOME_RECORD_MAGIC) &
				(ZeroHomeState[33]$UDINT <> 0);
			adminHomeIdentityValid :=
				(ZeroHomeState[1]$UDINT = adminDiagnosticsBuild) &
				(ZeroHomeState[2]$UDINT = adminBootId) &
				(ZeroHomeState[3]$UDINT = adminMapRevision) &
				(ZeroHomeState[4]$UDINT = adminOriginalRequestId) &
				(ZeroHomeState[5]$UDINT = adminClientIntentId0) &
				(ZeroHomeState[6]$UDINT = adminClientIntentId1) &
				(ZeroHomeState[7]$UDINT = adminClientIntentId2) &
				(ZeroHomeState[8]$UDINT = adminClientIntentId3) &
				(ZeroHomeState[9] = TO_DINT(Reference)) &
				(ZeroHomeState[10] = TO_DINT(adminHomeSemanticMode)) &
				(ZeroHomeState[11] = adminHomeExpectedActualPosition) &
				(ZeroHomeState[12] = adminHomeTargetPosition);
			adminHomeTerminal :=
				(ZeroHomeState[0] >= LMC_HOME_RECORD_SUCCEEDED) &
				(ZeroHomeState[0] <= LMC_HOME_RECORD_QUARANTINED);
			adminHomeStateConsistent := FALSE;
			if ZeroHomeState[0] = LMC_HOME_RECORD_RUNNING then
				adminHomeStateConsistent :=
					(ZeroHomeState[39] >= LMC_HOME_ENGINE_WAIT_RT) &
					(ZeroHomeState[39] <= LMC_HOME_ENGINE_FINALIZE) &
					(ZeroHomeState[34]$UDINT <> 0) &
					(ZeroHomeState[35]$UDINT <> 0) &
					(ZeroHomeState[36]$UDINT <> 0) &
					(ZeroHomeState[37]$UDINT <> 0) &
					(ZeroHomeState[38]$UDINT = adminHomeAxisMask) &
					(OwnershipState[7]$UDINT = ZeroHomeState[34]$UDINT) &
					(OwnershipState[8]$UDINT = ZeroHomeState[35]$UDINT) &
					(OwnershipState[9]$UDINT = ZeroHomeState[38]$UDINT);
			elsif adminHomeTerminal then
				adminHomeStateConsistent :=
					(ZeroHomeState[39] = LMC_HOME_ENGINE_TERMINAL) &
					(ZeroHomeState[57] = ZeroHomeState[0]) &
					((ZeroHomeState[56]$UDINT and
					  LMC_HOME_FLAG_OWNER_FINALIZE_ACCEPTED) <> 0) &
					((ZeroHomeState[56]$UDINT and
					  LMC_HOME_FLAG_TERMINAL_PUBLISHED) <> 0) &
					((ZeroHomeState[47] = 0) | (ZeroHomeState[47] = 1)) &
					((ZeroHomeState[0] = LMC_HOME_RECORD_QUARANTINED) |
					 ((ZeroHomeState[56]$UDINT and
					   LMC_HOME_FLAG_PREEMPTION_CLEANUP) <> 0) |
					 (ZeroHomeState[47] = 1)) &
					((ZeroHomeState[0] = LMC_HOME_RECORD_QUARANTINED) |
					 ((ZeroHomeState[56]$UDINT and
					   LMC_HOME_FLAG_EXACT_RT_TERMINAL) <> 0)) &
					((ZeroHomeState[0] = LMC_HOME_RECORD_QUARANTINED) |
					 ((ZeroHomeState[56]$UDINT and
					   LMC_HOME_FLAG_PREEMPTION_CLEANUP) <> 0) |
					 ((ZeroHomeState[60]$UDINT =
					   LMC_HOME_OWNER_RECEIPT_MAGIC) &
					  (ZeroHomeState[61] =
					   LMC_HOME_OWNER_RECEIPT_COMPLETE) &
					  (ZeroHomeState[62] = 0) &
					  (ZeroHomeState[63]$UDINT =
					   ZeroHomeState[33]$UDINT)));
				case ZeroHomeState[0] of
					LMC_HOME_RECORD_SUCCEEDED:
						adminHomeStateConsistent := adminHomeStateConsistent &
							(ZeroHomeState[58] =
							 LMC_OWNER_REPORT_TERMINAL_SUCCESS);
					LMC_HOME_RECORD_FAILED, LMC_HOME_RECORD_ABORTED:
						adminHomeStateConsistent := adminHomeStateConsistent &
							(ZeroHomeState[58] =
							 LMC_OWNER_REPORT_TERMINAL_SAFE_FAILURE);
					LMC_HOME_RECORD_QUARANTINED:
						adminHomeStateConsistent := adminHomeStateConsistent &
							(ZeroHomeState[58] = LMC_OWNER_REPORT_QUARANTINE);
				else
					adminHomeStateConsistent := FALSE;
				end_case;
			end_if;

			if RequestSize <> 56 then
				adminDetailCode := 5;
			elsif (Reference < 1) | (Reference > 4) then
				adminDetailCode := 4;
			elsif adminSchemaVersion <> 1 then
				adminDetailCode := 1;
			elsif adminRequestFlags <> 0 then
				adminDetailCode := 2;
			elsif adminRequestId = 0 then
				adminDetailCode := 3;
			elsif adminDiagnosticsBuild = 0 then
				adminDetailCode := 16;
			elsif (adminBootId = 0) | (adminCurrentBootId = 0) then
				adminDetailCode := 17;
			elsif adminMapRevision = 0 then
				adminDetailCode := 18;
			elsif (adminHomeSemanticMode <> 1) |
			      (adminHomeReserved <> 0) |
			      (adminHomeTargetPosition <> 0) then
				adminDetailCode := 36;
			elsif (OwnershipState[3]$UDINT <> 0) &
			      (adminCurrentBootId <> OwnershipState[3]$UDINT) then
				adminDetailCode := 17;
			elsif ZeroHomeState[0] = LMC_HOME_RECORD_EMPTY then
				adminDetailCode := 33;
			elsif adminHomeRecordValid = FALSE then
				adminDetailCode := 35;
			elsif adminHomeIdentityValid = FALSE then
				adminDetailCode := 36;
			elsif ((ZeroHomeState[0] <> LMC_HOME_RECORD_RUNNING) &
			       (adminHomeTerminal = FALSE)) |
			      (adminHomeStateConsistent = FALSE) then
				adminDetailCode := 35;
			end_if;

			if adminDetailCode = 0 then
				_memset(dest:=pResponseFrame, usByte:=0, cntr:=152);
				pResponseFrame^$UINT := 0;
				(pResponseFrame + 2)^$UINT := 144;
				(pResponseFrame + 4)^$UDINT := 0;
				(pResponseFrame + 8)^$UINT := 1;
				(pResponseFrame + 10)^$UINT := 0;
				(pResponseFrame + 12)^$UINT := 0;
				(pResponseFrame + 14)^$INT := 0;
				(pResponseFrame + 16)^$UDINT := adminRequestId;
				(pResponseFrame + 20)^$UDINT := 0;
				(pResponseFrame + 24)^$UINT := ZeroHomeState[0]$UINT;
				(pResponseFrame + 26)^$UINT := ZeroHomeState[10]$UINT;
				(pResponseFrame + 28)^$UDINT := ZeroHomeState[1]$UDINT;
				(pResponseFrame + 32)^$UDINT := ZeroHomeState[2]$UDINT;
				(pResponseFrame + 36)^$UDINT := ZeroHomeState[3]$UDINT;
				(pResponseFrame + 40)^$UDINT := ZeroHomeState[4]$UDINT;
				(pResponseFrame + 44)^$UDINT := ZeroHomeState[5]$UDINT;
				(pResponseFrame + 48)^$UDINT := ZeroHomeState[6]$UDINT;
				(pResponseFrame + 52)^$UDINT := ZeroHomeState[7]$UDINT;
				(pResponseFrame + 56)^$UDINT := ZeroHomeState[8]$UDINT;
				(pResponseFrame + 60)^$UINT := ZeroHomeState[9]$UINT;
				(pResponseFrame + 62)^$UINT := 0;
				(pResponseFrame + 64)^$DINT := ZeroHomeState[11];
				(pResponseFrame + 68)^$DINT := ZeroHomeState[12];
				(pResponseFrame + 72)^$UDINT := ZeroHomeState[13]$UDINT;
				(pResponseFrame + 76)^$UINT := ZeroHomeState[14]$UINT;
				(pResponseFrame + 78)^$INT := ZeroHomeState[15]$INT;
				(pResponseFrame + 80)^$UDINT := ZeroHomeState[16]$UDINT;
				(pResponseFrame + 84)^$UDINT := ZeroHomeState[17]$UDINT;
				(pResponseFrame + 88)^$DINT := ZeroHomeState[18];
				(pResponseFrame + 92)^$DINT := ZeroHomeState[19];
				(pResponseFrame + 96)^$DINT := ZeroHomeState[20];
				(pResponseFrame + 100)^$DINT := ZeroHomeState[21];
				(pResponseFrame + 104)^$DINT := ZeroHomeState[22];
				(pResponseFrame + 108)^$DINT := ZeroHomeState[23];
				(pResponseFrame + 112)^$DINT := ZeroHomeState[24];
				(pResponseFrame + 116)^$DINT := ZeroHomeState[25];
				(pResponseFrame + 120)^$DINT := ZeroHomeState[26];
				(pResponseFrame + 124)^$UDINT := ZeroHomeState[27]$UDINT;
				(pResponseFrame + 128)^$UDINT := ZeroHomeState[28]$UDINT;
				(pResponseFrame + 132)^$UDINT := ZeroHomeState[29]$UDINT;
				(pResponseFrame + 136)^$UDINT := ZeroHomeState[30]$UDINT;
				(pResponseFrame + 140)^$UDINT := ZeroHomeState[31]$UDINT;
				(pResponseFrame + 144)^$UDINT := ZeroHomeState[32]$UDINT;
				(pResponseFrame + 148)^$UDINT := ZeroHomeState[33]$UDINT;
				ResponseSize := 152;
			else
				_memset(dest:=pResponseFrame, usByte:=0, cntr:=24);
				pResponseFrame^$UINT := 0;
				(pResponseFrame + 2)^$UINT := 16;
				(pResponseFrame + 4)^$UDINT := 0;
				(pResponseFrame + 8)^$UINT := 1;
				(pResponseFrame + 10)^$UINT := 0;
				(pResponseFrame + 12)^$UINT := 1;
				(pResponseFrame + 14)^$INT := -31000;
				(pResponseFrame + 16)^$UDINT := adminRequestId;
				(pResponseFrame + 20)^$UDINT := adminDetailCode;
				ResponseSize := 24;
			end_if;

		0x7D19:
			if ResponseCapacity < 152 then
				RETURN;
			end_if;
			adminDetailCode := 0;
			adminSchemaVersion := 0;
			adminRequestFlags := 0;
			adminRequestId := 0;
			adminDiagnosticsBuild := 0;
			adminBootId := 0;
			adminMapRevision := 0;
			adminCurrentBootId := 0;
			adminOriginalRequestId := 0;
			adminClientIntentId0 := 0;
			adminClientIntentId1 := 0;
			adminClientIntentId2 := 0;
			adminClientIntentId3 := 0;
			adminHomeSemanticMode := 0;
			adminHomeReserved := 0;
			adminHomeExpectedActualPosition := 0;
			adminHomeTargetPosition := 0;
			adminHomeRecordGeneration := 0;
			if RequestSize >= 8 then
				adminSchemaVersion := pRequest^$UINT;
				adminRequestFlags := (pRequest + 2)^$UINT;
				adminRequestId := (pRequest + 4)^$UDINT;
			end_if;
			if RequestSize >= 60 then
				adminDiagnosticsBuild := (pRequest + 8)^$UDINT;
				adminBootId := (pRequest + 12)^$UDINT;
				adminMapRevision := (pRequest + 16)^$UDINT;
				adminCurrentBootId := (pRequest + 20)^$UDINT;
				adminOriginalRequestId := (pRequest + 24)^$UDINT;
				adminClientIntentId0 := (pRequest + 28)^$UDINT;
				adminClientIntentId1 := (pRequest + 32)^$UDINT;
				adminClientIntentId2 := (pRequest + 36)^$UDINT;
				adminClientIntentId3 := (pRequest + 40)^$UDINT;
				adminHomeSemanticMode := (pRequest + 44)^$UINT;
				adminHomeReserved := (pRequest + 46)^$UINT;
				adminHomeExpectedActualPosition := (pRequest + 48)^$DINT;
				adminHomeTargetPosition := (pRequest + 52)^$DINT;
				adminHomeRecordGeneration := (pRequest + 56)^$UDINT;
			end_if;
			adminHomeRecordValid :=
				(ZeroHomeState[51]$UDINT = LMC_HOME_RECORD_MAGIC) &
				(ZeroHomeState[33]$UDINT <> 0);
			adminHomeIdentityValid :=
				(ZeroHomeState[1]$UDINT = adminDiagnosticsBuild) &
				(ZeroHomeState[2]$UDINT = adminBootId) &
				(ZeroHomeState[3]$UDINT = adminMapRevision) &
				(ZeroHomeState[4]$UDINT = adminOriginalRequestId) &
				(ZeroHomeState[5]$UDINT = adminClientIntentId0) &
				(ZeroHomeState[6]$UDINT = adminClientIntentId1) &
				(ZeroHomeState[7]$UDINT = adminClientIntentId2) &
				(ZeroHomeState[8]$UDINT = adminClientIntentId3) &
				(ZeroHomeState[9] = TO_DINT(Reference)) &
				(ZeroHomeState[10] = TO_DINT(adminHomeSemanticMode)) &
				(ZeroHomeState[11] = adminHomeExpectedActualPosition) &
				(ZeroHomeState[12] = adminHomeTargetPosition);
			adminHomeTerminal :=
				(ZeroHomeState[0] >= LMC_HOME_RECORD_SUCCEEDED) &
				(ZeroHomeState[0] <= LMC_HOME_RECORD_QUARANTINED);

			if RequestSize <> 60 then
				adminDetailCode := 5;
			elsif (Reference < 1) | (Reference > 4) then
				adminDetailCode := 4;
			elsif adminSchemaVersion <> 1 then
				adminDetailCode := 1;
			elsif adminRequestFlags <> 0 then
				adminDetailCode := 2;
			elsif adminRequestId = 0 then
				adminDetailCode := 3;
			elsif (adminBootId = 0) | (adminCurrentBootId = 0) then
				adminDetailCode := 17;
			elsif (OwnershipState[3]$UDINT <> 0) &
			      (adminCurrentBootId <> OwnershipState[3]$UDINT) then
				adminDetailCode := 17;
			elsif ZeroHomeState[0] = LMC_HOME_RECORD_EMPTY then
				adminDetailCode := 33;
			elsif adminHomeRecordValid = FALSE then
				adminDetailCode := 35;
			elsif adminHomeIdentityValid = FALSE then
				adminDetailCode := 36;
			elsif adminHomeRecordGeneration <> ZeroHomeState[33]$UDINT then
				adminDetailCode := 36;
			elsif adminHomeTerminal = FALSE then
				adminDetailCode := 34;
			elsif (ZeroHomeState[39] <> LMC_HOME_ENGINE_TERMINAL) |
			      ((ZeroHomeState[56]$UDINT and
			        LMC_HOME_FLAG_OWNER_FINALIZE_ACCEPTED) = 0) |
			      ((ZeroHomeState[56]$UDINT and
			        LMC_HOME_FLAG_TERMINAL_PUBLISHED) = 0) |
			      ((ZeroHomeState[47] <> 0) & (ZeroHomeState[47] <> 1)) |
			      (((ZeroHomeState[0] <> LMC_HOME_RECORD_QUARANTINED) &
			        ((ZeroHomeState[56]$UDINT and
			          LMC_HOME_FLAG_PREEMPTION_CLEANUP) = 0)) &
			       (ZeroHomeState[47] <> 1)) |
			      ((ZeroHomeState[0] <> LMC_HOME_RECORD_QUARANTINED) &
			       ((ZeroHomeState[56]$UDINT and
			         LMC_HOME_FLAG_EXACT_RT_TERMINAL) = 0)) |
			      (((ZeroHomeState[0] <> LMC_HOME_RECORD_QUARANTINED) &
			        ((ZeroHomeState[56]$UDINT and
			          LMC_HOME_FLAG_PREEMPTION_CLEANUP) = 0)) &
			       ((ZeroHomeState[60]$UDINT <>
			         LMC_HOME_OWNER_RECEIPT_MAGIC) |
			        (ZeroHomeState[61] <>
			         LMC_HOME_OWNER_RECEIPT_COMPLETE) |
			        (ZeroHomeState[62] <> 0) |
			        (ZeroHomeState[63]$UDINT <>
			         ZeroHomeState[33]$UDINT))) then
				adminDetailCode := 34;
			end_if;

			if adminDetailCode = 0 then
				_memset(dest:=pResponseFrame, usByte:=0, cntr:=152);
				pResponseFrame^$UINT := 0;
				(pResponseFrame + 2)^$UINT := 144;
				(pResponseFrame + 4)^$UDINT := 0;
				(pResponseFrame + 8)^$UINT := 1;
				(pResponseFrame + 10)^$UINT := 0;
				(pResponseFrame + 12)^$UINT := 0;
				(pResponseFrame + 14)^$INT := 0;
				(pResponseFrame + 16)^$UDINT := adminRequestId;
				(pResponseFrame + 20)^$UDINT := 0;
				(pResponseFrame + 24)^$UINT := ZeroHomeState[0]$UINT;
				(pResponseFrame + 26)^$UINT := ZeroHomeState[10]$UINT;
				(pResponseFrame + 28)^$UDINT := ZeroHomeState[1]$UDINT;
				(pResponseFrame + 32)^$UDINT := ZeroHomeState[2]$UDINT;
				(pResponseFrame + 36)^$UDINT := ZeroHomeState[3]$UDINT;
				(pResponseFrame + 40)^$UDINT := ZeroHomeState[4]$UDINT;
				(pResponseFrame + 44)^$UDINT := ZeroHomeState[5]$UDINT;
				(pResponseFrame + 48)^$UDINT := ZeroHomeState[6]$UDINT;
				(pResponseFrame + 52)^$UDINT := ZeroHomeState[7]$UDINT;
				(pResponseFrame + 56)^$UDINT := ZeroHomeState[8]$UDINT;
				(pResponseFrame + 60)^$UINT := ZeroHomeState[9]$UINT;
				(pResponseFrame + 62)^$UINT := 0;
				(pResponseFrame + 64)^$DINT := ZeroHomeState[11];
				(pResponseFrame + 68)^$DINT := ZeroHomeState[12];
				(pResponseFrame + 72)^$UDINT := ZeroHomeState[13]$UDINT;
				(pResponseFrame + 76)^$UINT := ZeroHomeState[14]$UINT;
				(pResponseFrame + 78)^$INT := ZeroHomeState[15]$INT;
				(pResponseFrame + 80)^$UDINT := ZeroHomeState[16]$UDINT;
				(pResponseFrame + 84)^$UDINT := ZeroHomeState[17]$UDINT;
				(pResponseFrame + 88)^$DINT := ZeroHomeState[18];
				(pResponseFrame + 92)^$DINT := ZeroHomeState[19];
				(pResponseFrame + 96)^$DINT := ZeroHomeState[20];
				(pResponseFrame + 100)^$DINT := ZeroHomeState[21];
				(pResponseFrame + 104)^$DINT := ZeroHomeState[22];
				(pResponseFrame + 108)^$DINT := ZeroHomeState[23];
				(pResponseFrame + 112)^$DINT := ZeroHomeState[24];
				(pResponseFrame + 116)^$DINT := ZeroHomeState[25];
				(pResponseFrame + 120)^$DINT := ZeroHomeState[26];
				(pResponseFrame + 124)^$UDINT := ZeroHomeState[27]$UDINT;
				(pResponseFrame + 128)^$UDINT := ZeroHomeState[28]$UDINT;
				(pResponseFrame + 132)^$UDINT := ZeroHomeState[29]$UDINT;
				(pResponseFrame + 136)^$UDINT := ZeroHomeState[30]$UDINT;
				(pResponseFrame + 140)^$UDINT := ZeroHomeState[31]$UDINT;
				(pResponseFrame + 144)^$UDINT := ZeroHomeState[32]$UDINT;
				(pResponseFrame + 148)^$UDINT := ZeroHomeState[33]$UDINT;
				ZeroHomeState[48] := 1;
				ZeroHomeState[49]$UDINT := adminHomeRecordGeneration;
				ResponseSize := 152;
			else
				_memset(dest:=pResponseFrame, usByte:=0, cntr:=24);
				pResponseFrame^$UINT := 0;
				(pResponseFrame + 2)^$UINT := 16;
				(pResponseFrame + 4)^$UDINT := 0;
				(pResponseFrame + 8)^$UINT := 1;
				(pResponseFrame + 10)^$UINT := 0;
				(pResponseFrame + 12)^$UINT := 1;
				(pResponseFrame + 14)^$INT := -31000;
				(pResponseFrame + 16)^$UDINT := adminRequestId;
				(pResponseFrame + 20)^$UDINT := adminDetailCode;
				ResponseSize := 24;
			end_if;

	else
		ResponseSize := -1;
	end_case;

END_FUNCTION

FUNCTION GLOBAL LMCControlCommandService::ValidateAxisOwnershipIdentity
	VAR_INPUT
		CommandId 	: UINT;
		Reference 	: UINT;
		ExpectedAxisMask 	: UDINT;
		OwnerKind 	: UINT;
		ResourceKind 	: UINT;
		AdmissionMode 	: UINT;
		CallerSessionEpoch 	: UDINT;
		RequestSequence 	: UDINT;
		AdmissionToken 	: UDINT;
		OwnerGeneration 	: UDINT;
		RequiredPhase 	: UINT;
		pIdentity 	: ^void;
		IdentitySize 	: UDINT;
	END_VAR
	VAR_OUTPUT
		Result 	: DINT;
	END_VAR
	VAR
		axisIndex : DINT;
		axisBit : UDINT;
		referenceAxisMask : UDINT;
		recordBase : DINT;
		identityHeaderBase : DINT;
		identityCompareResult : UDINT;
		identityPrefixSize : UDINT;
		identityTailSize : UDINT;
		identityTailOffset : UDINT;
		identityPackedCommand : UDINT;
		identityPackedOwner : UDINT;
		pIdentityBytes : ^USINT;
		expectedState : DINT;
		resourceValid : BOOL;
		tupleValid : BOOL;
	END_VAR

	Result := -1;
	if (ExpectedAxisMask = 0) |
	   (ExpectedAxisMask > LMC_OWNER_ROBOT_AXIS_MASK) |
	   (AdmissionToken = 0) | (OwnerGeneration = 0) |
	   (CallerSessionEpoch = 0) | (RequestSequence = 0) |
	   (IdentitySize = 0) | (IdentitySize > 1320) |
	   (pIdentity = NIL) |
	   ((RequiredPhase <> LMC_OWNER_PHASE_RESERVED) &
	    (RequiredPhase <> LMC_OWNER_PHASE_ACTIVE) &
	    (RequiredPhase <> LMC_OWNER_PHASE_SESSION_CLOSED_ROLLBACK)) then
		RETURN;
	end_if;
	Result := ValidateAxisOwnership(
		CommandId:=CommandId,
		Reference:=Reference,
		ExpectedAxisMask:=ExpectedAxisMask,
		OwnerKind:=OwnerKind,
		ResourceKind:=ResourceKind,
		AdmissionMode:=AdmissionMode,
		CallerSessionEpoch:=CallerSessionEpoch,
		RequestSequence:=RequestSequence,
		AdmissionToken:=AdmissionToken,
		OwnerGeneration:=OwnerGeneration,
		RequiredPhase:=RequiredPhase);
	if Result <> 0 then
		RETURN;
	end_if;
	referenceAxisMask := 0;
	case Reference of
		1: referenceAxisMask := 0x00000001;
		2: referenceAxisMask := 0x00000002;
		3: referenceAxisMask := 0x00000004;
		4: referenceAxisMask := 0x00000008;
		5: referenceAxisMask := 0x00000010;
		6: referenceAxisMask := 0x00000020;
		7: referenceAxisMask := 0x00000040;
		8: referenceAxisMask := 0x00000080;
		9: referenceAxisMask := 0x00000100;
	else
	end_case;
	tupleValid := FALSE;
	case CommandId of
		0x2022:
			tupleValid :=
				(OwnerKind = LMC_OWNER_KIND_DIRECT) &
				(ResourceKind = LMC_OWNER_RESOURCE_AXIS) &
				(AdmissionMode = LMC_OWNER_ADMISSION_SAFETY) &
				(referenceAxisMask <> 0) &
				(ExpectedAxisMask <= LMC_OWNER_ROBOT_AXIS_MASK) &
				((ExpectedAxisMask and referenceAxisMask) <> 0);
		0x2023:
			tupleValid :=
				(OwnerKind = LMC_OWNER_KIND_DIRECT) &
				(ResourceKind = LMC_OWNER_RESOURCE_AXIS) &
				(referenceAxisMask <> 0) &
				(((AdmissionMode = LMC_OWNER_ADMISSION_ORDINARY) &
				  (ExpectedAxisMask = referenceAxisMask)) |
				 ((AdmissionMode = LMC_OWNER_ADMISSION_SAFETY) &
				  (ExpectedAxisMask <= LMC_OWNER_ROBOT_AXIS_MASK) &
				  ((ExpectedAxisMask and referenceAxisMask) <> 0)));
		0x2024, 0x209F, 0x20A0, 0x20A2:
			tupleValid :=
				(OwnerKind = LMC_OWNER_KIND_DIRECT) &
				(ResourceKind = LMC_OWNER_RESOURCE_AXIS) &
				(AdmissionMode = LMC_OWNER_ADMISSION_ORDINARY) &
				(referenceAxisMask <> 0) &
				(ExpectedAxisMask = referenceAxisMask);
		0x2047, 0x20A4, 0x7D22:
			tupleValid :=
				(OwnerKind = LMC_OWNER_KIND_GROUP) &
				(ResourceKind = LMC_OWNER_RESOURCE_AXIS) &
				(AdmissionMode = LMC_OWNER_ADMISSION_ORDINARY) &
				(Reference = 0x0100) &
				(ExpectedAxisMask = LMC_OWNER_PROFILE_AXIS_MASK);
		0x2048:
			tupleValid :=
				(OwnerKind = LMC_OWNER_KIND_GROUP) &
				(ResourceKind = LMC_OWNER_RESOURCE_AXIS) &
				(AdmissionMode = LMC_OWNER_ADMISSION_SAFETY) &
				(Reference = 0x0100) &
				(ExpectedAxisMask = LMC_OWNER_PROFILE_AXIS_MASK);
		0x2085:
			tupleValid :=
				(OwnerKind = LMC_OWNER_KIND_GROUP) &
				(ResourceKind = LMC_OWNER_RESOURCE_AXIS) &
				(AdmissionMode = LMC_OWNER_ADMISSION_SAFETY) &
				(Reference = 0x0100) &
				((ExpectedAxisMask = LMC_OWNER_PROFILE_AXIS_MASK) |
				 (ExpectedAxisMask = LMC_OWNER_ROBOT_AXIS_MASK));
		0x2049, 0x204A:
			tupleValid :=
				(OwnerKind = LMC_OWNER_KIND_GROUP) &
				(ResourceKind = LMC_OWNER_RESOURCE_AXIS) &
				(AdmissionMode = LMC_OWNER_ADMISSION_ORDINARY) &
				(Reference = 0x0100) &
				(ExpectedAxisMask = LMC_OWNER_ROBOT_AXIS_MASK);
		0x204B:
			tupleValid :=
				(OwnerKind = LMC_OWNER_KIND_GROUP) &
				(ResourceKind = LMC_OWNER_RESOURCE_AXIS) &
				(AdmissionMode = LMC_OWNER_ADMISSION_SAFETY) &
				(Reference = 0x0100) &
				(ExpectedAxisMask = LMC_OWNER_ROBOT_AXIS_MASK);
		0x20E7:
			tupleValid :=
				(OwnerKind = LMC_OWNER_KIND_GROUP) &
				(ResourceKind = LMC_OWNER_RESOURCE_AXIS) &
				(AdmissionMode = LMC_OWNER_ADMISSION_LIFECYCLE) &
				(Reference = 0x0100) &
				(ExpectedAxisMask = LMC_OWNER_ROBOT_AXIS_MASK);
		0x7D13:
			tupleValid :=
				(OwnerKind = LMC_OWNER_KIND_LMC_HOME) &
				(ResourceKind = LMC_OWNER_RESOURCE_LMC_HOME_ENGINE) &
				(AdmissionMode = LMC_OWNER_ADMISSION_LIFECYCLE) &
				(referenceAxisMask <> 0) &
				(referenceAxisMask <= 0x00000008) &
				(ExpectedAxisMask = referenceAxisMask);
		0x7D15:
			tupleValid :=
				(OwnerKind = LMC_OWNER_KIND_DS402_HOME) &
				(ResourceKind = LMC_OWNER_RESOURCE_DS402_HOME_ENGINE) &
				(AdmissionMode = LMC_OWNER_ADMISSION_LIFECYCLE) &
				(referenceAxisMask <> 0) &
				(referenceAxisMask <= 0x00000008) &
				(ExpectedAxisMask = referenceAxisMask);
		0x7E53:
			tupleValid :=
				(OwnerKind = LMC_OWNER_KIND_ENCODER) &
				(ResourceKind = LMC_OWNER_RESOURCE_DIAGNOSTICS_SDO_ENGINE) &
				(AdmissionMode = LMC_OWNER_ADMISSION_LIFECYCLE) &
				(referenceAxisMask <> 0) &
				(referenceAxisMask <= 0x00000008) &
				(ExpectedAxisMask = referenceAxisMask);
	else
	end_case;
	if tupleValid = FALSE then
		RETURN;
	end_if;
	expectedState := LMC_OWNER_STATE_RESERVED;
	if RequiredPhase = LMC_OWNER_PHASE_SESSION_CLOSED_ROLLBACK then
		if (CommandId <> 0x7D15) |
		   (OwnerKind <> LMC_OWNER_KIND_DS402_HOME) |
		   (ResourceKind <> LMC_OWNER_RESOURCE_DS402_HOME_ENGINE) |
		   (AdmissionMode <> LMC_OWNER_ADMISSION_LIFECYCLE) then
			RETURN;
		end_if;
		expectedState := LMC_OWNER_STATE_QUARANTINED;
	elsif RequiredPhase = LMC_OWNER_PHASE_ACTIVE then
		if AdmissionMode = LMC_OWNER_ADMISSION_SAFETY then
			if (OwnerKind = LMC_OWNER_KIND_DIRECT) |
			   (OwnerKind = LMC_OWNER_KIND_GROUP) then
				expectedState := LMC_OWNER_STATE_SAFETY_PREEMPTING;
			else
				RETURN;
			end_if;
		else
			case OwnerKind of
				LMC_OWNER_KIND_DIRECT:
					expectedState := LMC_OWNER_STATE_DIRECT_ACTIVE;
				LMC_OWNER_KIND_GROUP:
					expectedState := LMC_OWNER_STATE_GROUP_ACTIVE;
				LMC_OWNER_KIND_LMC_HOME:
					expectedState := LMC_OWNER_STATE_LMC_HOME_ACTIVE;
				LMC_OWNER_KIND_DS402_HOME:
					expectedState := LMC_OWNER_STATE_DS402_HOME_ACTIVE;
				LMC_OWNER_KIND_ENCODER:
					expectedState := LMC_OWNER_STATE_TW20_QUEUED;
			else
				RETURN;
			end_case;
		end_if;
	end_if;
	if (OwnershipState[0]$UDINT <> LMC_OWNER_TABLE_MAGIC) |
	   (OwnershipState[3]$UDINT = 0) |
	   (OwnershipState[24] <> 0) then
		Result := -3;
		RETURN;
	end_if;

	resourceValid :=
		(ResourceKind = LMC_OWNER_RESOURCE_AXIS) &
		(OwnershipState[7]$UDINT <> AdmissionToken) &
		(OwnershipState[8]$UDINT <> OwnerGeneration) &
		(OwnershipState[10]$UDINT <> AdmissionToken) &
		(OwnershipState[11]$UDINT <> OwnerGeneration) &
		(OwnershipState[13]$UDINT <> AdmissionToken) &
		(OwnershipState[14]$UDINT <> OwnerGeneration);
	case ResourceKind of
		LMC_OWNER_RESOURCE_LMC_HOME_ENGINE:
			resourceValid :=
				(OwnershipState[7]$UDINT = AdmissionToken) &
				(OwnershipState[8]$UDINT = OwnerGeneration) &
				(OwnershipState[9]$UDINT = ExpectedAxisMask);
		LMC_OWNER_RESOURCE_DS402_HOME_ENGINE:
			resourceValid :=
				(OwnershipState[10]$UDINT = AdmissionToken) &
				(OwnershipState[11]$UDINT = OwnerGeneration) &
				(OwnershipState[12]$UDINT = ExpectedAxisMask);
		LMC_OWNER_RESOURCE_DIAGNOSTICS_SDO_ENGINE:
			resourceValid :=
				(OwnershipState[13]$UDINT = AdmissionToken) &
				(OwnershipState[14]$UDINT = OwnerGeneration) &
				(OwnershipState[15]$UDINT = ExpectedAxisMask);
	else
	end_case;
	if resourceValid = FALSE then
		Result := -2;
		RETURN;
	end_if;

	axisIndex := 1;
	while axisIndex <= LMC_OWNER_AXIS_COUNT do
		case axisIndex of
			1: axisBit := 0x00000001;
			2: axisBit := 0x00000002;
			3: axisBit := 0x00000004;
			4: axisBit := 0x00000008;
			5: axisBit := 0x00000010;
			6: axisBit := 0x00000020;
			7: axisBit := 0x00000040;
			8: axisBit := 0x00000080;
			9: axisBit := 0x00000100;
		else
			axisBit := 0;
		end_case;
		recordBase := LMC_OWNER_GLOBAL_SLOTS +
			((axisIndex - 1) * LMC_OWNER_AXIS_STRIDE);
		if (ExpectedAxisMask and axisBit) <> 0 then
			if (OwnershipState[recordBase + 1] =
			    LMC_OWNER_STATE_QUARANTINED) &
			   (RequiredPhase <>
			    LMC_OWNER_PHASE_SESSION_CLOSED_ROLLBACK) then
				Result := -3;
				RETURN;
			elsif (OwnershipState[recordBase] <> axisIndex) |
			      (OwnershipState[recordBase + 35]$UDINT <>
			       (LMC_OWNER_AXIS_RECORD_MAGIC + TO_UDINT(axisIndex))) |
			      (OwnershipState[recordBase + 1] <> expectedState) |
			      (OwnershipState[recordBase + 2] <> TO_DINT(OwnerKind)) |
			      (OwnershipState[recordBase + 3] <> TO_DINT(CommandId)) |
			      (OwnershipState[recordBase + 4]$UDINT <> AdmissionToken) |
			      (OwnershipState[recordBase + 5]$UDINT <> OwnerGeneration) |
			      (OwnershipState[recordBase + 6]$UDINT <>
			       CallerSessionEpoch) |
			      (OwnershipState[recordBase + 7]$UDINT <> RequestSequence) |
			      (OwnershipState[recordBase + 11]$UDINT <>
			       ExpectedAxisMask) |
			      (OwnershipState[recordBase + 12] <> TO_DINT(Reference)) |
			      (OwnershipState[recordBase + 13] <>
			       TO_DINT(ResourceKind)) |
			      (OwnershipState[recordBase + 14] <>
			       TO_DINT(AdmissionMode)) then
				Result := -2;
				RETURN;
			end_if;
		elsif (OwnershipState[recordBase + 4]$UDINT = AdmissionToken) |
		      (OwnershipState[recordBase + 5]$UDINT = OwnerGeneration) then
			Result := -2;
			RETURN;
		end_if;
		axisIndex += 1;
	end_while;
	pIdentityBytes := pIdentity$^USINT;
	identityPrefixSize := IdentitySize;
	if identityPrefixSize > LMC_OWNER_IDENTITY_PREFIX_BYTES then
		identityPrefixSize := LMC_OWNER_IDENTITY_PREFIX_BYTES;
	end_if;
	identityTailSize := 0;
	if IdentitySize > LMC_OWNER_IDENTITY_PREFIX_BYTES then
		identityTailSize := IdentitySize - LMC_OWNER_IDENTITY_PREFIX_BYTES;
	end_if;
	identityTailOffset := 0;
	if OwnerKind <> LMC_OWNER_KIND_GROUP then
		identityTailOffset := TO_UDINT(Reference - 1) * 8;
		if identityTailSize > 8 then
			Result := -1;
			RETURN;
		end_if;
	end_if;
	identityPackedCommand := TO_UDINT(CommandId) or
		(TO_UDINT(Reference) shl 16);
	identityPackedOwner := TO_UDINT(OwnerKind) or
		(TO_UDINT(ResourceKind) shl 8) or
		(TO_UDINT(AdmissionMode) shl 16);
	axisIndex := 1;
	while axisIndex <= LMC_OWNER_AXIS_COUNT do
		case axisIndex of
			1: axisBit := 0x00000001;
			2: axisBit := 0x00000002;
			3: axisBit := 0x00000004;
			4: axisBit := 0x00000008;
			5: axisBit := 0x00000010;
			6: axisBit := 0x00000020;
			7: axisBit := 0x00000040;
			8: axisBit := 0x00000080;
			9: axisBit := 0x00000100;
		else
			axisBit := 0;
		end_case;
		if (ExpectedAxisMask and axisBit) <> 0 then
			recordBase := LMC_OWNER_GLOBAL_SLOTS +
				((axisIndex - 1) * LMC_OWNER_AXIS_STRIDE);
			if OwnershipState[recordBase + 15]$UDINT <> IdentitySize then
				Result := -2;
				RETURN;
			end_if;
			if OwnerKind = LMC_OWNER_KIND_GROUP then
				identityHeaderBase := LMC_OWNER_IDENTITY_GROUP_HEADER_BASE;
				if (OwnershipIdentityState[identityHeaderBase]$UDINT <>
				    LMC_OWNER_IDENTITY_GROUP_MAGIC) |
				   (OwnershipIdentityState[identityHeaderBase + 1] <>
				    LMC_OWNER_IDENTITY_VERSION) |
				   (OwnershipIdentityState[identityHeaderBase + 2]$UDINT <>
				    IdentitySize) |
				   (OwnershipIdentityState[identityHeaderBase + 3]$UDINT <>
				    AdmissionToken) |
				   (OwnershipIdentityState[identityHeaderBase + 4]$UDINT <>
				    OwnerGeneration) |
				   (OwnershipIdentityState[identityHeaderBase + 5]$UDINT <>
				    ExpectedAxisMask) |
				   (OwnershipIdentityState[identityHeaderBase + 6]$UDINT <>
				    CallerSessionEpoch) |
				   (OwnershipIdentityState[identityHeaderBase + 7]$UDINT <>
				    RequestSequence) |
				   (OwnershipIdentityState[identityHeaderBase + 8]$UDINT <>
				    identityPackedCommand) |
				   (OwnershipIdentityState[identityHeaderBase + 9]$UDINT <>
				    identityPackedOwner) then
					Result := -3;
					RETURN;
				end_if;
			else
				identityHeaderBase := LMC_OWNER_IDENTITY_AXIS_HEADER_BASE +
					((axisIndex - 1) *
					 LMC_OWNER_IDENTITY_AXIS_HEADER_STRIDE);
				if (OwnershipIdentityState[identityHeaderBase]$UDINT <>
				    (LMC_OWNER_IDENTITY_AXIS_MAGIC + TO_UDINT(axisIndex))) |
				   (OwnershipIdentityState[identityHeaderBase + 1] <>
				    LMC_OWNER_IDENTITY_VERSION) |
				   (OwnershipIdentityState[identityHeaderBase + 2]$UDINT <>
				    IdentitySize) |
				   (OwnershipIdentityState[identityHeaderBase + 3]$UDINT <>
				    AdmissionToken) |
				   (OwnershipIdentityState[identityHeaderBase + 4]$UDINT <>
				    OwnerGeneration) |
				   (OwnershipIdentityState[identityHeaderBase + 5]$UDINT <>
				    ExpectedAxisMask) |
				   (OwnershipIdentityState[identityHeaderBase + 6]$UDINT <>
				    CallerSessionEpoch) |
				   (OwnershipIdentityState[identityHeaderBase + 7]$UDINT <>
				    RequestSequence) |
				   (OwnershipIdentityState[identityHeaderBase + 8]$UDINT <>
				    identityPackedCommand) |
				   (OwnershipIdentityState[identityHeaderBase + 9]$UDINT <>
				    identityPackedOwner) |
				   (OwnershipIdentityState[identityHeaderBase + 10]$UDINT <>
				    identityTailOffset) |
				   (OwnershipIdentityState[identityHeaderBase + 11]$UDINT <>
				    identityTailSize) then
					Result := -3;
					RETURN;
				end_if;
			end_if;
			identityCompareResult := _memcmp(
				ptr1:=#OwnershipState[recordBase + 16],
				ptr2:=pIdentityBytes, cntr:=identityPrefixSize);
			if identityCompareResult <> 0 then
				Result := -2;
				RETURN;
			end_if;
			if identityTailSize > 0 then
				identityCompareResult := _memcmp(
					ptr1:=#OwnershipIdentityState[
					 TO_DINT(identityTailOffset / 4)],
					ptr2:=pIdentityBytes +
					 LMC_OWNER_IDENTITY_PREFIX_BYTES,
					cntr:=identityTailSize);
				if identityCompareResult <> 0 then
					Result := -2;
					RETURN;
				end_if;
			end_if;
		end_if;
		axisIndex += 1;
	end_while;
	Result := 0;

END_FUNCTION

FUNCTION GLOBAL LMCControlCommandService::CopyAxisOwnershipPreemption
	VAR_INPUT
		PreemptedAdmissionToken 	: UDINT;
		PreemptedOwnerGeneration 	: UDINT;
		pDest 	: ^void;
		DestSize 	: UDINT;
	END_VAR
	VAR_OUTPUT
		Result 	: DINT;
	END_VAR
	VAR
		axisIndex : DINT;
		axisBit : UDINT;
		recordBase : DINT;
		firstRecordBase : DINT;
		currentRecordBase : DINT;
		safetyRecordBase : DINT;
		identityHeaderBase : DINT;
		identityCompareResult : UDINT;
		stateIndex : DINT;
		oldAxisMask : UDINT;
		oldToken : UDINT;
		oldGeneration : UDINT;
		oldSession : UDINT;
		oldSequence : UDINT;
		oldCommand : DINT;
		oldReference : DINT;
		oldOwnerKind : DINT;
		oldResourceKind : DINT;
		oldAdmissionMode : DINT;
		oldState : DINT;
		identitySize : UDINT;
		identityExpectedSize : UDINT;
		identityPrefixSize : UDINT;
		identityTailSize : UDINT;
		identityTailOffset : UDINT;
		identityPackedCommand : UDINT;
		identityPackedOwner : UDINT;
		totalSize : UDINT;
		preemptFlags : UDINT;
		cleanupRequiredMask : UDINT;
		cleanupCompleteMask : UDINT;
		safetyAxisMask : UDINT;
		safetyToken : UDINT;
		safetyGeneration : UDINT;
		safetyCommand : UDINT;
		safetyReference : UDINT;
		safetyReferenceAxisMask : UDINT;
		safetyOwnerKind : DINT;
		safetyResourceKind : DINT;
		safetyState : DINT;
		safetySession : UDINT;
		safetySequence : UDINT;
		safetyAdmission : DINT;
		referenceAxisMask : UDINT;
		pDestBytes : ^USINT;
		bankDirty : BOOL;
		oldFound : BOOL;
		tupleValid : BOOL;
		identityMetadataValid : BOOL;
		disjointCurrentValid : BOOL;
		currentStateValid : BOOL;
		safetyFound : BOOL;
	END_VAR

	Result := -1;
	if (PreemptedAdmissionToken = 0) |
	   (PreemptedOwnerGeneration = 0) | (pDest = NIL) then
		RETURN;
	end_if;
	pDestBytes := pDest$^USINT;
	if DestSize < LMC_OWNER_PREEMPT_COPY_HEADER_BYTES then
		Result := -4;
		RETURN;
	end_if;
	_memset(dest:=pDestBytes, usByte:=0,
		cntr:=LMC_OWNER_PREEMPT_COPY_HEADER_BYTES);

	if OwnershipPreemptedIdentityState[
	   LMC_OWNER_PREEMPT_HEADER_BASE]$UDINT <>
	   LMC_OWNER_PREEMPT_IDENTITY_MAGIC then
		bankDirty := FALSE;
		stateIndex := 0;
		while stateIndex <= 323 do
			if OwnershipPreemptedState[stateIndex] <> 0 then
				bankDirty := TRUE;
			end_if;
			stateIndex += 1;
		end_while;
		stateIndex := 0;
		while stateIndex <= 431 do
			if OwnershipPreemptedIdentityState[stateIndex] <> 0 then
				bankDirty := TRUE;
			end_if;
			stateIndex += 1;
		end_while;
		if bankDirty then
			OwnershipState[24] := 1;
			Result := -3;
		else
			Result := LMC_OWNER_PREEMPT_STATUS_NONE;
		end_if;
		RETURN;
	end_if;
	preemptFlags := OwnershipPreemptedIdentityState[
		LMC_OWNER_PREEMPT_HEADER_BASE + 1]$UDINT;
	cleanupRequiredMask := OwnershipPreemptedIdentityState[
		LMC_OWNER_PREEMPT_HEADER_BASE + 8]$UDINT;
	cleanupCompleteMask := OwnershipPreemptedIdentityState[
		LMC_OWNER_PREEMPT_HEADER_BASE + 9]$UDINT;
	safetyToken := OwnershipPreemptedIdentityState[
		LMC_OWNER_PREEMPT_HEADER_BASE + 2]$UDINT;
	safetyGeneration := OwnershipPreemptedIdentityState[
		LMC_OWNER_PREEMPT_HEADER_BASE + 3]$UDINT;
	safetyAxisMask := OwnershipPreemptedIdentityState[
		LMC_OWNER_PREEMPT_HEADER_BASE + 4]$UDINT;
	safetySession := OwnershipPreemptedIdentityState[
		LMC_OWNER_PREEMPT_HEADER_BASE + 5]$UDINT;
	safetySequence := OwnershipPreemptedIdentityState[
		LMC_OWNER_PREEMPT_HEADER_BASE + 6]$UDINT;
	safetyCommand := OwnershipPreemptedIdentityState[
		LMC_OWNER_PREEMPT_HEADER_BASE + 7]$UDINT and 0x0000FFFF;
	safetyReference := (OwnershipPreemptedIdentityState[
		LMC_OWNER_PREEMPT_HEADER_BASE + 7]$UDINT shr 16) and 0x0000FFFF;
	if ((preemptFlags and 0x0000FFFF) <>
	    LMC_OWNER_IDENTITY_VERSION) |
	   ((preemptFlags and 0xFFFE0000) <> 0) |
	   (safetyToken = 0) | (safetyGeneration = 0) |
	   (safetySession = 0) | (safetySequence = 0) |
	   (safetyAxisMask = 0) |
	   (safetyAxisMask > LMC_OWNER_ROBOT_AXIS_MASK) |
	   ((cleanupRequiredMask and (not safetyAxisMask)) <> 0) |
	   ((cleanupCompleteMask and (not cleanupRequiredMask)) <> 0) then
		OwnershipState[24] := 1;
		Result := -3;
		RETURN;
	end_if;
	safetyReferenceAxisMask := 0;
	case safetyReference of
		1: safetyReferenceAxisMask := 0x00000001;
		2: safetyReferenceAxisMask := 0x00000002;
		3: safetyReferenceAxisMask := 0x00000004;
		4: safetyReferenceAxisMask := 0x00000008;
		5: safetyReferenceAxisMask := 0x00000010;
		6: safetyReferenceAxisMask := 0x00000020;
		7: safetyReferenceAxisMask := 0x00000040;
		8: safetyReferenceAxisMask := 0x00000080;
		9: safetyReferenceAxisMask := 0x00000100;
	else
	end_case;
	safetyOwnerKind := 0;
	safetyResourceKind := LMC_OWNER_RESOURCE_AXIS;
	case safetyCommand of
		0x2022, 0x2023:
			if (safetyReferenceAxisMask <> 0) &
			   ((safetyAxisMask and safetyReferenceAxisMask) <> 0) then
				safetyOwnerKind := LMC_OWNER_KIND_DIRECT;
			end_if;
		0x2048:
			if (safetyReference = 0x0100) &
			   (safetyAxisMask = LMC_OWNER_PROFILE_AXIS_MASK) then
				safetyOwnerKind := LMC_OWNER_KIND_GROUP;
			end_if;
		0x2085:
			if (safetyReference = 0x0100) &
			   ((safetyAxisMask = LMC_OWNER_PROFILE_AXIS_MASK) |
			    (safetyAxisMask = LMC_OWNER_ROBOT_AXIS_MASK)) then
				safetyOwnerKind := LMC_OWNER_KIND_GROUP;
			end_if;
		0x204B:
			if (safetyReference = 0x0100) &
			   (safetyAxisMask = LMC_OWNER_ROBOT_AXIS_MASK) then
				safetyOwnerKind := LMC_OWNER_KIND_GROUP;
			end_if;
	else
	end_case;
	if safetyOwnerKind = 0 then
		OwnershipState[24] := 1;
		Result := -3;
		RETURN;
	end_if;

	oldFound := FALSE;
	tupleValid := TRUE;
	firstRecordBase := -1;
	axisIndex := 1;
	while axisIndex <= LMC_OWNER_AXIS_COUNT do
		recordBase := (axisIndex - 1) * LMC_OWNER_AXIS_STRIDE;
		if (OwnershipPreemptedState[recordBase] <> axisIndex) |
		   (OwnershipPreemptedState[recordBase + 35]$UDINT <>
		    (LMC_OWNER_AXIS_RECORD_MAGIC + TO_UDINT(axisIndex))) then
			tupleValid := FALSE;
		elsif (OwnershipPreemptedState[recordBase + 4]$UDINT =
		       PreemptedAdmissionToken) &
		      (OwnershipPreemptedState[recordBase + 5]$UDINT =
		       PreemptedOwnerGeneration) then
			if oldFound = FALSE then
				oldAxisMask := OwnershipPreemptedState[recordBase + 11]$UDINT;
				oldToken := OwnershipPreemptedState[recordBase + 4]$UDINT;
				oldGeneration := OwnershipPreemptedState[recordBase + 5]$UDINT;
				oldSession := OwnershipPreemptedState[recordBase + 6]$UDINT;
				oldSequence := OwnershipPreemptedState[recordBase + 7]$UDINT;
				oldCommand := OwnershipPreemptedState[recordBase + 3];
				oldReference := OwnershipPreemptedState[recordBase + 12];
				oldOwnerKind := OwnershipPreemptedState[recordBase + 2];
				oldResourceKind := OwnershipPreemptedState[recordBase + 13];
				oldAdmissionMode := OwnershipPreemptedState[recordBase + 14];
				oldState := OwnershipPreemptedState[recordBase + 1];
				identitySize := OwnershipPreemptedState[recordBase + 15]$UDINT;
				oldFound := TRUE;
			else
				if (oldAxisMask <>
				    OwnershipPreemptedState[recordBase + 11]$UDINT) |
				   (oldSession <>
				    OwnershipPreemptedState[recordBase + 6]$UDINT) |
				   (oldSequence <>
				    OwnershipPreemptedState[recordBase + 7]$UDINT) |
				   (oldCommand <> OwnershipPreemptedState[recordBase + 3]) |
				   (oldReference <> OwnershipPreemptedState[recordBase + 12]) |
				   (oldOwnerKind <> OwnershipPreemptedState[recordBase + 2]) |
				   (oldResourceKind <> OwnershipPreemptedState[recordBase + 13]) |
				   (oldAdmissionMode <> OwnershipPreemptedState[recordBase + 14]) |
				   (oldState <> OwnershipPreemptedState[recordBase + 1]) |
				   (identitySize <>
				    OwnershipPreemptedState[recordBase + 15]$UDINT) then
					tupleValid := FALSE;
				end_if;
			end_if;
		elsif (OwnershipPreemptedState[recordBase + 4]$UDINT =
		       PreemptedAdmissionToken) |
		      (OwnershipPreemptedState[recordBase + 5]$UDINT =
		       PreemptedOwnerGeneration) then
			tupleValid := FALSE;
		end_if;
		axisIndex += 1;
	end_while;
	if oldFound = FALSE then
		Result := -2;
		RETURN;
	end_if;
	if (tupleValid = FALSE) | (oldAxisMask = 0) |
	   (oldAxisMask > LMC_OWNER_ROBOT_AXIS_MASK) |
	   (oldToken = 0) | (oldGeneration = 0) |
	   (oldSession = 0) | (oldSequence = 0) |
	   (identitySize = 0) | (identitySize > 1320) then
		OwnershipState[24] := 1;
		Result := -3;
		RETURN;
	end_if;

	// The compact preemption bank does not retain the old identity header.
	// Reconstruct and validate every header field available in the exact record
	// snapshot before copying the preserved prefix and suffix bytes.
	referenceAxisMask := 0;
	case oldReference of
		1: referenceAxisMask := 0x00000001;
		2: referenceAxisMask := 0x00000002;
		3: referenceAxisMask := 0x00000004;
		4: referenceAxisMask := 0x00000008;
		5: referenceAxisMask := 0x00000010;
		6: referenceAxisMask := 0x00000020;
		7: referenceAxisMask := 0x00000040;
		8: referenceAxisMask := 0x00000080;
		9: referenceAxisMask := 0x00000100;
	else
	end_case;
	identityExpectedSize := 0;
	identityMetadataValid := FALSE;
	case oldCommand of
		0x2022:
			identityExpectedSize := 16;
			identityMetadataValid :=
				(oldOwnerKind = LMC_OWNER_KIND_DIRECT) &
				(oldResourceKind = LMC_OWNER_RESOURCE_AXIS) &
				(oldAdmissionMode = LMC_OWNER_ADMISSION_SAFETY) &
				(referenceAxisMask <> 0) &
				((oldAxisMask and referenceAxisMask) <> 0);
		0x2023:
			identityExpectedSize := 8;
			identityMetadataValid :=
				(oldOwnerKind = LMC_OWNER_KIND_DIRECT) &
				(oldResourceKind = LMC_OWNER_RESOURCE_AXIS) &
				(referenceAxisMask <> 0) &
				(((oldAdmissionMode = LMC_OWNER_ADMISSION_ORDINARY) &
				  (oldAxisMask = referenceAxisMask)) |
				 ((oldAdmissionMode = LMC_OWNER_ADMISSION_SAFETY) &
				  ((oldAxisMask and referenceAxisMask) <> 0)));
		0x2024:
			identityExpectedSize := 1;
			identityMetadataValid :=
				(oldOwnerKind = LMC_OWNER_KIND_DIRECT) &
				(oldResourceKind = LMC_OWNER_RESOURCE_AXIS) &
				(oldAdmissionMode = LMC_OWNER_ADMISSION_ORDINARY) &
				(referenceAxisMask <> 0) &
				(oldAxisMask = referenceAxisMask);
		0x209F, 0x20A0:
			identityExpectedSize := 32;
			identityMetadataValid :=
				(oldOwnerKind = LMC_OWNER_KIND_DIRECT) &
				(oldResourceKind = LMC_OWNER_RESOURCE_AXIS) &
				(oldAdmissionMode = LMC_OWNER_ADMISSION_ORDINARY) &
				(referenceAxisMask <> 0) &
				(oldAxisMask = referenceAxisMask);
		0x20A2:
			identityExpectedSize := 24;
			identityMetadataValid :=
				(oldOwnerKind = LMC_OWNER_KIND_DIRECT) &
				(oldResourceKind = LMC_OWNER_RESOURCE_AXIS) &
				(oldAdmissionMode = LMC_OWNER_ADMISSION_ORDINARY) &
				(referenceAxisMask <> 0) &
				(oldAxisMask = referenceAxisMask);
		0x2047:
			identityExpectedSize := 1;
			identityMetadataValid :=
				(oldOwnerKind = LMC_OWNER_KIND_GROUP) &
				(oldResourceKind = LMC_OWNER_RESOURCE_AXIS) &
				(oldAdmissionMode = LMC_OWNER_ADMISSION_ORDINARY) &
				(oldReference = 0x0100) &
				(oldAxisMask = LMC_OWNER_PROFILE_AXIS_MASK);
		0x20A4:
			identityExpectedSize := 96;
			identityMetadataValid :=
				(oldOwnerKind = LMC_OWNER_KIND_GROUP) &
				(oldResourceKind = LMC_OWNER_RESOURCE_AXIS) &
				(oldAdmissionMode = LMC_OWNER_ADMISSION_ORDINARY) &
				(oldReference = 0x0100) &
				(oldAxisMask = LMC_OWNER_PROFILE_AXIS_MASK);
		0x7D22:
			identityExpectedSize := 104;
			identityMetadataValid :=
				(oldOwnerKind = LMC_OWNER_KIND_GROUP) &
				(oldResourceKind = LMC_OWNER_RESOURCE_AXIS) &
				(oldAdmissionMode = LMC_OWNER_ADMISSION_ORDINARY) &
				(oldReference = 0x0100) &
				(oldAxisMask = LMC_OWNER_PROFILE_AXIS_MASK);
		0x2048:
			identityExpectedSize := 1;
			identityMetadataValid :=
				(oldOwnerKind = LMC_OWNER_KIND_GROUP) &
				(oldResourceKind = LMC_OWNER_RESOURCE_AXIS) &
				(oldAdmissionMode = LMC_OWNER_ADMISSION_SAFETY) &
				(oldReference = 0x0100) &
				(oldAxisMask = LMC_OWNER_PROFILE_AXIS_MASK);
		0x2085:
			identityExpectedSize := 16;
			identityMetadataValid :=
				(oldOwnerKind = LMC_OWNER_KIND_GROUP) &
				(oldResourceKind = LMC_OWNER_RESOURCE_AXIS) &
				(oldAdmissionMode = LMC_OWNER_ADMISSION_SAFETY) &
				(oldReference = 0x0100) &
				((oldAxisMask = LMC_OWNER_PROFILE_AXIS_MASK) |
				 (oldAxisMask = LMC_OWNER_ROBOT_AXIS_MASK));
		0x2049, 0x204A:
			identityExpectedSize := 1;
			identityMetadataValid :=
				(oldOwnerKind = LMC_OWNER_KIND_GROUP) &
				(oldResourceKind = LMC_OWNER_RESOURCE_AXIS) &
				(oldAdmissionMode = LMC_OWNER_ADMISSION_ORDINARY) &
				(oldReference = 0x0100) &
				(oldAxisMask = LMC_OWNER_ROBOT_AXIS_MASK);
		0x204B:
			identityExpectedSize := 1;
			identityMetadataValid :=
				(oldOwnerKind = LMC_OWNER_KIND_GROUP) &
				(oldResourceKind = LMC_OWNER_RESOURCE_AXIS) &
				(oldAdmissionMode = LMC_OWNER_ADMISSION_SAFETY) &
				(oldReference = 0x0100) &
				(oldAxisMask = LMC_OWNER_ROBOT_AXIS_MASK);
		0x20E7:
			identityExpectedSize := 1320;
			identityMetadataValid :=
				(oldOwnerKind = LMC_OWNER_KIND_GROUP) &
				(oldResourceKind = LMC_OWNER_RESOURCE_AXIS) &
				(oldAdmissionMode = LMC_OWNER_ADMISSION_LIFECYCLE) &
				(oldReference = 0x0100) &
				(oldAxisMask = LMC_OWNER_ROBOT_AXIS_MASK);
		0x7D13:
			identityExpectedSize := 56;
			identityMetadataValid :=
				(oldOwnerKind = LMC_OWNER_KIND_LMC_HOME) &
				(oldResourceKind = LMC_OWNER_RESOURCE_LMC_HOME_ENGINE) &
				(oldAdmissionMode = LMC_OWNER_ADMISSION_LIFECYCLE) &
				(referenceAxisMask <> 0) &
				(referenceAxisMask <= 0x00000008) &
				(oldAxisMask = referenceAxisMask);
		0x7D15:
			identityExpectedSize := 72;
			identityMetadataValid :=
				(oldOwnerKind = LMC_OWNER_KIND_DS402_HOME) &
				(oldResourceKind = LMC_OWNER_RESOURCE_DS402_HOME_ENGINE) &
				(oldAdmissionMode = LMC_OWNER_ADMISSION_LIFECYCLE) &
				(referenceAxisMask <> 0) &
				(referenceAxisMask <= 0x00000008) &
				(oldAxisMask = referenceAxisMask);
		0x7E53:
			identityExpectedSize := 72;
			identityMetadataValid :=
				(oldOwnerKind = LMC_OWNER_KIND_ENCODER) &
				(oldResourceKind =
				 LMC_OWNER_RESOURCE_DIAGNOSTICS_SDO_ENGINE) &
				(oldAdmissionMode = LMC_OWNER_ADMISSION_LIFECYCLE) &
				(referenceAxisMask <> 0) &
				(referenceAxisMask <= 0x00000008) &
				(oldAxisMask = referenceAxisMask);
	else
	end_case;
	if oldState <> LMC_OWNER_STATE_QUARANTINED then
		case oldOwnerKind of
			LMC_OWNER_KIND_DIRECT:
				identityMetadataValid := identityMetadataValid &
					((oldState = LMC_OWNER_STATE_RESERVED) |
					 (oldState = LMC_OWNER_STATE_DIRECT_ACTIVE));
			LMC_OWNER_KIND_GROUP:
				identityMetadataValid := identityMetadataValid &
					((oldState = LMC_OWNER_STATE_RESERVED) |
					 (oldState = LMC_OWNER_STATE_GROUP_LEASE) |
					 (oldState = LMC_OWNER_STATE_GROUP_ACTIVE));
			LMC_OWNER_KIND_LMC_HOME:
				identityMetadataValid := identityMetadataValid &
					((oldState = LMC_OWNER_STATE_RESERVED) |
					 (oldState = LMC_OWNER_STATE_LMC_HOME_ACTIVE));
			LMC_OWNER_KIND_DS402_HOME:
				identityMetadataValid := identityMetadataValid &
					((oldState = LMC_OWNER_STATE_RESERVED) |
					 (oldState = LMC_OWNER_STATE_DS402_HOME_ACTIVE));
			LMC_OWNER_KIND_ENCODER:
				identityMetadataValid := identityMetadataValid &
					((oldState = LMC_OWNER_STATE_RESERVED) |
					 (oldState = LMC_OWNER_STATE_TW20_QUEUED) |
					 (oldState = LMC_OWNER_STATE_TW20_RUNNING) |
					 (oldState = LMC_OWNER_STATE_TW20_DRAINING));
		else
			identityMetadataValid := FALSE;
		end_case;
	end_if;
	if (identityMetadataValid = FALSE) |
	   (identitySize <> identityExpectedSize) then
		OwnershipState[24] := 1;
		Result := -3;
		RETURN;
	end_if;
	identityPackedCommand := TO_UDINT(oldCommand) or
		(TO_UDINT(oldReference) shl 16);
	identityPackedOwner := TO_UDINT(oldOwnerKind) or
		(TO_UDINT(oldResourceKind) shl 8) or
		(TO_UDINT(oldAdmissionMode) shl 16);
	identityPrefixSize := identitySize;
	if identityPrefixSize > LMC_OWNER_IDENTITY_PREFIX_BYTES then
		identityPrefixSize := LMC_OWNER_IDENTITY_PREFIX_BYTES;
	end_if;
	identityTailSize := 0;
	if identitySize > LMC_OWNER_IDENTITY_PREFIX_BYTES then
		identityTailSize := identitySize - LMC_OWNER_IDENTITY_PREFIX_BYTES;
	end_if;
	identityTailOffset := 0;
	if oldOwnerKind <> LMC_OWNER_KIND_GROUP then
		identityTailOffset := TO_UDINT(oldReference - 1) * 8;
	end_if;
	if ((oldOwnerKind <> LMC_OWNER_KIND_GROUP) &
	    (identityTailSize > 8)) |
	   ((identityTailOffset + identityTailSize) >
	    LMC_OWNER_IDENTITY_SUFFIX_BYTES) then
		OwnershipState[24] := 1;
		Result := -3;
		RETURN;
	end_if;
	axisIndex := 1;
	while axisIndex <= LMC_OWNER_AXIS_COUNT do
		case axisIndex of
			1: axisBit := 0x00000001;
			2: axisBit := 0x00000002;
			3: axisBit := 0x00000004;
			4: axisBit := 0x00000008;
			5: axisBit := 0x00000010;
			6: axisBit := 0x00000020;
			7: axisBit := 0x00000040;
			8: axisBit := 0x00000080;
			9: axisBit := 0x00000100;
		else
			axisBit := 0;
		end_case;
		recordBase := (axisIndex - 1) * LMC_OWNER_AXIS_STRIDE;
		if (oldAxisMask and axisBit) <> 0 then
			if (OwnershipPreemptedState[recordBase + 4]$UDINT <> oldToken) |
			   (OwnershipPreemptedState[recordBase + 5]$UDINT <>
			    oldGeneration) |
			   (OwnershipPreemptedState[recordBase + 6]$UDINT <> oldSession) |
			   (OwnershipPreemptedState[recordBase + 7]$UDINT <> oldSequence) |
			   (OwnershipPreemptedState[recordBase + 11]$UDINT <>
			    oldAxisMask) |
			   (OwnershipPreemptedState[recordBase + 15]$UDINT <>
			    identitySize) |
			   ((TO_UDINT(OwnershipPreemptedState[recordBase + 3]) or
			     (TO_UDINT(OwnershipPreemptedState[recordBase + 12]) shl 16)) <>
			    identityPackedCommand) |
			   ((TO_UDINT(OwnershipPreemptedState[recordBase + 2]) or
			     (TO_UDINT(OwnershipPreemptedState[recordBase + 13]) shl 8) or
			     (TO_UDINT(OwnershipPreemptedState[recordBase + 14]) shl 16)) <>
			    identityPackedOwner) then
				tupleValid := FALSE;
			end_if;
			if firstRecordBase < 0 then
				firstRecordBase := recordBase;
			else
				identityCompareResult := _memcmp(
					ptr1:=#OwnershipPreemptedState[firstRecordBase + 16],
					ptr2:=#OwnershipPreemptedState[recordBase + 16],
					cntr:=identityPrefixSize);
				if identityCompareResult <> 0 then
					tupleValid := FALSE;
				end_if;
			end_if;
		elsif (OwnershipPreemptedState[recordBase + 4]$UDINT = oldToken) |
		      (OwnershipPreemptedState[recordBase + 5]$UDINT =
		       oldGeneration) then
			tupleValid := FALSE;
		end_if;
		axisIndex += 1;
	end_while;
	if tupleValid = FALSE then
		OwnershipState[24] := 1;
		Result := -3;
		RETURN;
	end_if;
	if ((oldAxisMask and safetyAxisMask) <> 0) &
	   ((oldAxisMask and safetyAxisMask) <> oldAxisMask) then
		OwnershipState[24] := 1;
		Result := -3;
		RETURN;
	end_if;
	if (oldAxisMask and safetyAxisMask) = 0 then
		// The bank snapshots every axis. A disjoint old tuple was not
		// preempted; prove that its live immutable tuple and exact identity
		// still exist before returning the zero-header NONE result.
		disjointCurrentValid := TRUE;
		axisIndex := 1;
		while axisIndex <= LMC_OWNER_AXIS_COUNT do
			case axisIndex of
				1: axisBit := 0x00000001;
				2: axisBit := 0x00000002;
				3: axisBit := 0x00000004;
				4: axisBit := 0x00000008;
				5: axisBit := 0x00000010;
				6: axisBit := 0x00000020;
				7: axisBit := 0x00000040;
				8: axisBit := 0x00000080;
				9: axisBit := 0x00000100;
			else
				axisBit := 0;
			end_case;
			recordBase := (axisIndex - 1) * LMC_OWNER_AXIS_STRIDE;
			currentRecordBase := LMC_OWNER_GLOBAL_SLOTS + recordBase;
			if (oldAxisMask and axisBit) <> 0 then
				currentStateValid := FALSE;
				case oldOwnerKind of
					LMC_OWNER_KIND_DIRECT:
						currentStateValid :=
							OwnershipState[currentRecordBase + 1] =
							LMC_OWNER_STATE_DIRECT_ACTIVE;
					LMC_OWNER_KIND_GROUP:
						currentStateValid :=
							(OwnershipState[currentRecordBase + 1] =
							 LMC_OWNER_STATE_GROUP_LEASE) |
							(OwnershipState[currentRecordBase + 1] =
							 LMC_OWNER_STATE_GROUP_ACTIVE);
					LMC_OWNER_KIND_LMC_HOME:
						currentStateValid :=
							OwnershipState[currentRecordBase + 1] =
							LMC_OWNER_STATE_LMC_HOME_ACTIVE;
					LMC_OWNER_KIND_DS402_HOME:
						currentStateValid :=
							OwnershipState[currentRecordBase + 1] =
							LMC_OWNER_STATE_DS402_HOME_ACTIVE;
					LMC_OWNER_KIND_ENCODER:
						currentStateValid :=
							(OwnershipState[currentRecordBase + 1] =
							 LMC_OWNER_STATE_TW20_QUEUED) |
							(OwnershipState[currentRecordBase + 1] =
							 LMC_OWNER_STATE_TW20_RUNNING) |
							(OwnershipState[currentRecordBase + 1] =
							 LMC_OWNER_STATE_TW20_DRAINING);
				else
				end_case;
				if (OwnershipState[currentRecordBase] <> axisIndex) |
				   (OwnershipState[currentRecordBase + 35]$UDINT <>
				    (LMC_OWNER_AXIS_RECORD_MAGIC + TO_UDINT(axisIndex))) |
				   (OwnershipState[currentRecordBase + 2] <> oldOwnerKind) |
				   (OwnershipState[currentRecordBase + 3] <> oldCommand) |
				   (OwnershipState[currentRecordBase + 4]$UDINT <> oldToken) |
				   (OwnershipState[currentRecordBase + 5]$UDINT <>
				    oldGeneration) |
				   (OwnershipState[currentRecordBase + 6]$UDINT <> oldSession) |
				   (OwnershipState[currentRecordBase + 7]$UDINT <> oldSequence) |
				   (OwnershipState[currentRecordBase + 11]$UDINT <>
				    oldAxisMask) |
				   (OwnershipState[currentRecordBase + 12] <> oldReference) |
				   (OwnershipState[currentRecordBase + 13] <>
				    oldResourceKind) |
				   (OwnershipState[currentRecordBase + 14] <>
				    oldAdmissionMode) |
				   (OwnershipState[currentRecordBase + 15]$UDINT <>
				    identitySize) | (currentStateValid = FALSE) then
					disjointCurrentValid := FALSE;
				end_if;
				if oldOwnerKind = LMC_OWNER_KIND_GROUP then
					identityHeaderBase :=
						LMC_OWNER_IDENTITY_GROUP_HEADER_BASE;
					if (OwnershipIdentityState[identityHeaderBase]$UDINT <>
					    LMC_OWNER_IDENTITY_GROUP_MAGIC) |
					   (OwnershipIdentityState[identityHeaderBase + 1] <>
					    LMC_OWNER_IDENTITY_VERSION) |
					   (OwnershipIdentityState[identityHeaderBase + 2]$UDINT <>
					    identitySize) |
					   (OwnershipIdentityState[identityHeaderBase + 3]$UDINT <>
					    oldToken) |
					   (OwnershipIdentityState[identityHeaderBase + 4]$UDINT <>
					    oldGeneration) |
					   (OwnershipIdentityState[identityHeaderBase + 5]$UDINT <>
					    oldAxisMask) |
					   (OwnershipIdentityState[identityHeaderBase + 6]$UDINT <>
					    oldSession) |
					   (OwnershipIdentityState[identityHeaderBase + 7]$UDINT <>
					    oldSequence) |
					   (OwnershipIdentityState[identityHeaderBase + 8]$UDINT <>
					    identityPackedCommand) |
					   (OwnershipIdentityState[identityHeaderBase + 9]$UDINT <>
					    identityPackedOwner) then
						disjointCurrentValid := FALSE;
					end_if;
				else
					identityHeaderBase := LMC_OWNER_IDENTITY_AXIS_HEADER_BASE +
						((axisIndex - 1) *
						 LMC_OWNER_IDENTITY_AXIS_HEADER_STRIDE);
					if (OwnershipIdentityState[identityHeaderBase]$UDINT <>
					    (LMC_OWNER_IDENTITY_AXIS_MAGIC + TO_UDINT(axisIndex))) |
					   (OwnershipIdentityState[identityHeaderBase + 1] <>
					    LMC_OWNER_IDENTITY_VERSION) |
					   (OwnershipIdentityState[identityHeaderBase + 2]$UDINT <>
					    identitySize) |
					   (OwnershipIdentityState[identityHeaderBase + 3]$UDINT <>
					    oldToken) |
					   (OwnershipIdentityState[identityHeaderBase + 4]$UDINT <>
					    oldGeneration) |
					   (OwnershipIdentityState[identityHeaderBase + 5]$UDINT <>
					    oldAxisMask) |
					   (OwnershipIdentityState[identityHeaderBase + 6]$UDINT <>
					    oldSession) |
					   (OwnershipIdentityState[identityHeaderBase + 7]$UDINT <>
					    oldSequence) |
					   (OwnershipIdentityState[identityHeaderBase + 8]$UDINT <>
					    identityPackedCommand) |
					   (OwnershipIdentityState[identityHeaderBase + 9]$UDINT <>
					    identityPackedOwner) |
					   (OwnershipIdentityState[identityHeaderBase + 10]$UDINT <>
					    identityTailOffset) |
					   (OwnershipIdentityState[identityHeaderBase + 11]$UDINT <>
					    identityTailSize) then
						disjointCurrentValid := FALSE;
					end_if;
				end_if;
				identityCompareResult := _memcmp(
					ptr1:=#OwnershipState[currentRecordBase + 16],
					ptr2:=#OwnershipPreemptedState[recordBase + 16],
					cntr:=identityPrefixSize);
				if identityCompareResult <> 0 then
					disjointCurrentValid := FALSE;
				end_if;
				if identityTailSize > 0 then
					identityCompareResult := _memcmp(
						ptr1:=#OwnershipIdentityState[
						 TO_DINT(identityTailOffset / 4)],
						ptr2:=#OwnershipPreemptedIdentityState[
						 TO_DINT(identityTailOffset / 4)],
						cntr:=identityTailSize);
					if identityCompareResult <> 0 then
						disjointCurrentValid := FALSE;
					end_if;
				end_if;
			elsif (OwnershipState[currentRecordBase + 4]$UDINT = oldToken) |
			      (OwnershipState[currentRecordBase + 5]$UDINT =
			       oldGeneration) then
				disjointCurrentValid := FALSE;
			end_if;
			axisIndex += 1;
		end_while;
		if disjointCurrentValid = FALSE then
			OwnershipState[24] := 1;
			Result := -3;
		else
			Result := LMC_OWNER_PREEMPT_STATUS_NONE;
		end_if;
		RETURN;
	end_if;

	safetyFound := FALSE;
	tupleValid := TRUE;
	axisIndex := 1;
	while axisIndex <= LMC_OWNER_AXIS_COUNT do
		case axisIndex of
			1: axisBit := 0x00000001;
			2: axisBit := 0x00000002;
			3: axisBit := 0x00000004;
			4: axisBit := 0x00000008;
			5: axisBit := 0x00000010;
			6: axisBit := 0x00000020;
			7: axisBit := 0x00000040;
			8: axisBit := 0x00000080;
			9: axisBit := 0x00000100;
		else
			axisBit := 0;
		end_case;
		safetyRecordBase := LMC_OWNER_GLOBAL_SLOTS +
			((axisIndex - 1) * LMC_OWNER_AXIS_STRIDE);
		if (safetyAxisMask and axisBit) <> 0 then
			if (OwnershipState[safetyRecordBase] <> axisIndex) |
			   (OwnershipState[safetyRecordBase + 35]$UDINT <>
			    (LMC_OWNER_AXIS_RECORD_MAGIC + TO_UDINT(axisIndex))) |
			   (OwnershipState[safetyRecordBase + 2] <> safetyOwnerKind) |
			   (OwnershipState[safetyRecordBase + 3]$UDINT <> safetyCommand) |
			   (OwnershipState[safetyRecordBase + 4]$UDINT <> safetyToken) |
			   (OwnershipState[safetyRecordBase + 5]$UDINT <>
			    safetyGeneration) |
			   (OwnershipState[safetyRecordBase + 6]$UDINT <> safetySession) |
			   (OwnershipState[safetyRecordBase + 7]$UDINT <> safetySequence) |
			   (OwnershipState[safetyRecordBase + 11]$UDINT <>
			    safetyAxisMask) |
			   (OwnershipState[safetyRecordBase + 12]$UDINT <>
			    safetyReference) |
			   (OwnershipState[safetyRecordBase + 13] <>
			    safetyResourceKind) |
			   (OwnershipState[safetyRecordBase + 14] <>
			    LMC_OWNER_ADMISSION_SAFETY) then
				tupleValid := FALSE;
			elsif safetyFound = FALSE then
				safetyState := OwnershipState[safetyRecordBase + 1];
				safetyAdmission := OwnershipState[safetyRecordBase + 14];
				safetyFound := TRUE;
			elsif safetyState <> OwnershipState[safetyRecordBase + 1] then
				tupleValid := FALSE;
			end_if;
		elsif (OwnershipState[safetyRecordBase + 4]$UDINT = safetyToken) |
		      (OwnershipState[safetyRecordBase + 5]$UDINT =
		       safetyGeneration) then
			tupleValid := FALSE;
		end_if;
		axisIndex += 1;
	end_while;
	if (safetyFound = FALSE) | (tupleValid = FALSE) |
	   ((safetyState <> LMC_OWNER_STATE_RESERVED) &
	    (safetyState <> LMC_OWNER_STATE_SAFETY_PREEMPTING) &
	    (safetyState <> LMC_OWNER_STATE_QUARANTINED)) then
		OwnershipState[24] := 1;
		Result := -3;
		RETURN;
	end_if;

	if safetyState = LMC_OWNER_STATE_RESERVED then
		Result := LMC_OWNER_PREEMPT_STATUS_PENDING_FREEZE;
	elsif (preemptFlags and
	       LMC_OWNER_PREEMPT_FLAG_FORCE_QUARANTINE) <> 0 then
		Result := LMC_OWNER_PREEMPT_STATUS_CLEANUP_QUARANTINED;
	elsif (cleanupCompleteMask and cleanupRequiredMask) <>
	      cleanupRequiredMask then
		Result := LMC_OWNER_PREEMPT_STATUS_CLEANUP_REQUIRED;
	else
		Result := LMC_OWNER_PREEMPT_STATUS_CLEANUP_COMPLETE;
	end_if;
	totalSize := LMC_OWNER_PREEMPT_COPY_HEADER_BYTES + identitySize;
	if DestSize < totalSize then
		Result := -4;
		RETURN;
	end_if;
	(pDestBytes + 4)^$UDINT := LMC_OWNER_IDENTITY_VERSION;
	(pDestBytes + 8)^$UDINT := LMC_OWNER_PREEMPT_COPY_HEADER_BYTES;
	(pDestBytes + 12)^$UDINT := totalSize;
	(pDestBytes + 16)^$DINT := Result;
	(pDestBytes + 20)^$UDINT := preemptFlags and 0xFFFF0000;
	(pDestBytes + 24)^$UDINT := cleanupRequiredMask;
	(pDestBytes + 28)^$UDINT := cleanupCompleteMask;
	(pDestBytes + 32)^$UDINT := oldAxisMask;
	(pDestBytes + 36)^$UDINT := oldToken;
	(pDestBytes + 40)^$UDINT := oldGeneration;
	(pDestBytes + 44)^$UDINT := oldSession;
	(pDestBytes + 48)^$UDINT := oldSequence;
	(pDestBytes + 52)^$DINT := oldCommand;
	(pDestBytes + 56)^$DINT := oldReference;
	(pDestBytes + 60)^$DINT := oldOwnerKind;
	(pDestBytes + 64)^$DINT := oldResourceKind;
	(pDestBytes + 68)^$DINT := oldAdmissionMode;
	(pDestBytes + 72)^$DINT := oldState;
	(pDestBytes + 76)^$UDINT := identitySize;
	recordBase := 0;
	axisIndex := 1;
	while axisIndex <= LMC_OWNER_AXIS_COUNT do
		recordBase := (axisIndex - 1) * LMC_OWNER_AXIS_STRIDE;
		if (OwnershipPreemptedState[recordBase + 4]$UDINT = oldToken) &
		   (OwnershipPreemptedState[recordBase + 5]$UDINT =
		    oldGeneration) then
			exit;
		end_if;
		axisIndex += 1;
	end_while;
	(pDestBytes + 80)^$UDINT :=
		OwnershipPreemptedState[recordBase + 8]$UDINT;
	(pDestBytes + 84)^$UDINT :=
		OwnershipPreemptedState[recordBase + 9]$UDINT;
	(pDestBytes + 88)^$UDINT :=
		OwnershipPreemptedState[recordBase + 10]$UDINT;
	(pDestBytes + 92)^$DINT := OwnershipPreemptedState[recordBase + 32];
	(pDestBytes + 96)^$UDINT :=
		OwnershipPreemptedState[recordBase + 33]$UDINT;
	(pDestBytes + 100)^$UDINT :=
		OwnershipPreemptedState[recordBase + 34]$UDINT;
	(pDestBytes + 104)^$UDINT := safetyAxisMask;
	(pDestBytes + 108)^$UDINT := safetyToken;
	(pDestBytes + 112)^$UDINT := safetyGeneration;
	(pDestBytes + 116)^$UDINT := safetyCommand;
	(pDestBytes + 120)^$UDINT := safetyReference;
	(pDestBytes + 124)^$DINT := safetyState;
	(pDestBytes + 128)^$UDINT := safetySession;
	(pDestBytes + 132)^$UDINT := safetySequence;
	(pDestBytes + 136)^$DINT := safetyAdmission;
	(pDestBytes + 140)^$UDINT := 0;
	_memcpy(ptr1:=pDestBytes + LMC_OWNER_PREEMPT_COPY_HEADER_BYTES,
		ptr2:=#OwnershipPreemptedState[recordBase + 16],
		cntr:=identityPrefixSize);
	if identityTailSize > 0 then
		_memcpy(ptr1:=pDestBytes + LMC_OWNER_PREEMPT_COPY_HEADER_BYTES +
			identityPrefixSize,
			ptr2:=#OwnershipPreemptedIdentityState[
			 TO_DINT(identityTailOffset / 4)], cntr:=identityTailSize);
	end_if;
	pDestBytes^$UDINT := LMC_OWNER_PREEMPT_COPY_MAGIC;

END_FUNCTION

FUNCTION GLOBAL LMCControlCommandService::PublishAxisOwnershipPreemptionCleanup
	VAR_INPUT
		ExpectedAxisMask 	: UDINT;
		PreemptedAdmissionToken 	: UDINT;
		PreemptedOwnerGeneration 	: UDINT;
		SafetyAdmissionToken 	: UDINT;
		SafetyOwnerGeneration 	: UDINT;
		CleanupKind 	: UINT;
		ReportValue0 	: UDINT;
		ReportValue1 	: UDINT;
		ObservationCycle 	: UDINT;
	END_VAR
	VAR_OUTPUT
		Result 	: DINT;
	END_VAR
	VAR
		axisIndex : DINT;
		axisBit : UDINT;
		identityIndex : DINT;
		oldRecordBase : DINT;
		safetyRecordBase : DINT;
		firstSafetyRecordBase : DINT;
		evidenceRecordBase : DINT;
		observerBase : DINT;
		evidenceObserverBase : DINT;
		preemptObserverBase : DINT;
		identityHeaderBase : DINT;
		identityCompareResult : UDINT;
		preemptFlags : UDINT;
		cleanupRequiredMask : UDINT;
		cleanupCompleteMask : UDINT;
		safetyAxisMask : UDINT;
		safetySession : UDINT;
		safetySequence : UDINT;
		safetyPackedCommand : UDINT;
		safetyPackedOwner : UDINT;
		safetyIdentitySize : UDINT;
		safetyIdentityPrefixSize : UDINT;
		safetyIdentityTailOffset : UDINT;
		referenceAxisMask : UDINT;
		observerFlags : UDINT;
		oldAxisMask : UDINT;
		oldSession : UDINT;
		oldSequence : UDINT;
		oldIdentitySize : UDINT;
		oldIdentityExpectedSize : UDINT;
		oldIdentityPrefixSize : UDINT;
		oldIdentityTailSize : UDINT;
		oldIdentityTailOffset : UDINT;
		oldIdentityPackedCommand : UDINT;
		oldIdentityPackedOwner : UDINT;
		oldCommand : DINT;
		oldReference : DINT;
		oldOwnerKind : DINT;
		oldResourceKind : DINT;
		oldAdmissionMode : DINT;
		oldState : DINT;
		safetyCommand : DINT;
		safetyReference : DINT;
		safetyOwnerKind : DINT;
		safetyResourceKind : DINT;
		safetyAdmissionMode : DINT;
		safetyState : DINT;
		publishedCleanupKind : DINT;
		oldFound : BOOL;
		safetyFound : BOOL;
		tupleValid : BOOL;
		exactReplay : BOOL;
		replayEvidenceMatch : BOOL;
		cleanupAlreadyPublished : BOOL;
		publishedCleanupValid : BOOL;
		oldSpecialValid : BOOL;
		oldBankValid : BOOL;
		rootValid : BOOL;
		safetyEscalated : BOOL;
		safetyForceQuarantine : BOOL;
		safetyOverlayFound : BOOL;
		oldIdentityValid : BOOL;
		oldObserverValid : BOOL;
		safetyIdentityValid : BOOL;
		safetyObserverValid : BOOL;
	END_VAR
